//--------------------------------------------------------------------------------------
// Cyclic action
	IF (me.StateMachine.intState=me.StateMachine.intStateLastCycle) THEN
		
		//----------------------------------------------------------------------
		// Substates to let pass hanger(S) from zone 1
		// Triggered by command "Release" (common job interface)
		//----------------------------------------------------------------------		
		CASE me.SubStateMachine.intState OF	
			cSTA_SUB_WAIT_FOR_CMD:
				// Wait for command release
				IF (me.intCmd=STB_CmdState.cCMD_RELEASE) THEN
					CIf.Job.intACmd:=cSTA_DONE;
					me.SubStateMachine.intStateNext := cSTA_SUB_SEND_RELEASE;		
				END_IF
					
			cSTA_SUB_SEND_RELEASE:				
				// Send release command to buffer zone 1
				a_pBufferZoneChildCIF[0]^.Job.intACmd:= STB_CmdState.cCMD_RELEASE;
							
				// State Change Condition
				IF(a_pBufferZoneChildCIF[0]^.Job.intState = STB_CmdState.cSTA_RELEASE)THEN
					me.SubStateMachine.intStateNext := cSTA_SUB_SEND_STOP;					
				END_IF		

			cSTA_SUB_SEND_STOP:
				// Send stop command to buffer zone 1
				a_pBufferZoneChildCIF[0]^.Job.intACmd:= cCMD_STOP;	
				
				// State Change Condition
				IF(a_pBufferZoneChildCIF[0]^.Job.intState = cSTA_STOP)THEN
					me.SubStateMachine.intStateNext := cSTA_SUB_WAIT_FOR_CMD;																
				END_IF	
		
			cSTA_SUB_BREAK:
				//..not used	
		
		END_CASE
				
		
		//----------------------------------------------------------------------
		// Continuous refill of all zones
		//----------------------------------------------------------------------
		
		// Only execute method if more than one buffer zones exist!
		// Note: Slide buffer controller can also used with only one buffer.
		IF (usiNumOfBufferZones>1) THEN				
			THIS^.RefillZones();
		END_IF
			
			
		// Sub state machine general handling
		me.SubStateMachine.intStateLastCycle := me.SubStateMachine.intState;
		CIf.Job.strSubState := THIS^.getCmdState(intCmdState:=me.SubStateMachine.intState,bolState:=TRUE);
		IF (me.SubStateMachine.intState<>me.SubStateMachine.intStateNext) THEN
			me.SubStateMachine.intState := me.SubStateMachine.intStateNext;  // set next state for next cycle
			me.SubStateMachine.udiTimeInState_ms := 0; // reset timer
			// log state change -> open point
		ELSE
			// increment time in state	
			me.SubStateMachine.udiTimeInState_ms := me.SubStateMachine.udiTimeInState_ms + me.FUBInfo.udiSample_ms;
		END_IF
	
		
		// State Change Condition
		IF ((me.intCmd=cCMD_STOP) AND (me.SubStateMachine.intState=cSTA_SUB_WAIT_FOR_CMD))THEN
			me.StateMachine.intStateNext := cSTA_STOPBusy;
		ELSIF ((me.intCmd=STB_CmdState.cCMD_RELEASE_ALL) AND (me.SubStateMachine.intState=cSTA_SUB_WAIT_FOR_CMD))THEN
			me.StateMachine.intStateNext := STB_CmdState.cSTA_RELEASE_ALLBusy;
		END_IF
	END_IF

//--------------------------------------------------------------------------------------
// Exit action
	IF (me.StateMachine.intState<>me.StateMachine.intStateNext) THEN
		;
	END_IF
END_METHOD

METHOD PROTECTED sta_RUNBusy : BOOL
// state implemetation
//--------------------------------------------------------------------------------------
// Entry action
	IF (me.StateMachine.intState<>me.StateMachine.intStateLastCycle) THEN
		me.StateMachine.intStateLastCycle := me.StateMachine.intState;
		
		// Init for refill sequence
		intIndexRefill:= 0;
		SubStateMachineRefill:=0;
	
		// Initialize sub state machine
		me.SubStateMachine.intState:= cSTA_SUB_WAIT_FOR_CMD; 
		me.SubStateMachine.intStateNext := cSTA_SUB_WAIT_FOR_CMD;
	END_IF

	
//--------------------------------------------------------------------------------------
// Cyclic action
	IF (me.StateMachine.intState=me.StateMachine.intStateLastCycle) THEN
			
	
		// State Change Condition	
		IF (TRUE) THEN
			me.StateMachine.intStateNext := cSTA_RUN;		
		END_IF

	END_IF

//--------------------------------------------------------------------------------------
// Exit action
	IF (me.StateMachine.intState<>me.StateMachine.intStateNext) THEN
		;
	END_IF
END_METHOD

METHOD PROTECTED sta_STOP : BOOL
// state implemetation
//--------------------------------------------------------------------------------------
// Entry action
	IF (me.StateMachine.intState<>me.StateMachine.intStateLastCycle) THEN
		me.StateMachine.intStateLastCycle := me.StateMachine.intState;
		;
	END_IF

//--------------------------------------------------------------------------------------
// Cyclic action
	IF (me.StateMachine.intState=me.StateMachine.intStateLastCycle) THEN

	
		// State Change Condition	
		IF (me.intCmd = cCMD_RUN) THEN 
			me.StateMachine.intStateNext := cSTA_RUNBusy;
		ELSIF(me.intCmd = SLB_CmdState.cCMD_RELEASE_ALL) THEN
			me.StateMachine.intStateNext := SLB_CmdState.cSTA_RELEASE_ALLBusy;
		END_IF
	END_IF

//-------------------------------------------------------------------------------------
// Exit action
	IF (me.StateMachine.intState<>me.StateMachine.intStateNext) THEN
		;
	END_IF
END_METHOD

METHOD PROTECTED sta_STOPBusy : BOOL
// state implemetation
//--------------------------------------------------------------------------------------
// Entry action
	IF (me.StateMachine.intState<>me.StateMachine.intStateLastCycle) THEN
		me.StateMachine.intStateLastCycle := me.StateMachine.intState;
		
		// send command STOP to all existing buffer zone child controller.
		THIS^.CmdToAllZones(cCMD_STOP);

	END_IF

//--------------------------------------------------------------------------------------
// Cyclic action
	IF (me.StateMachine.intState=me.StateMachine.intStateLastCycle) THEN
			
				
		// State Change Condition
		// Check if all STOPPED
		IF (THIS^.checkStateAllZones(cSTA_STOP)) THEN
			me.StateMachine.intStateNext := cSTA_STOP;
		END_IF
	END_IF

//--------------------------------------------------------------------------------------
// Exit action
	IF (me.StateMachine.intState<>me.StateMachine.intStateNext) THEN
		;
	END_IF
END_METHOD

METHOD PROTECTED StateMachine : BOOL
SUPER^.StateMachine();

// main statemachine of base controller
CASE me.StateMachine.intState OF
    cSTA_STOPBusy: 
        THIS^.sta_STOPBusy();
    cSTA_STOP: 
        THIS^.sta_STOP();
	cSTA_RUNBusy: 
        THIS^.sta_RUNBusy();
    cSTA_RUN: 
        THIS^.sta_RUN();				
    SLB_CmdState.cSTA_RELEASE_ALLBusy: 
        THIS^.sta_RELEASE_ALLBusy();
    SLB_CmdState.cSTA_RELEASE_ALL: 
        THIS^.sta_RELEASE_ALL();
END_CASE;
END_METHOD

END_FUNCTION_BLOCK

// POUs/Controller/Lvl2/COS (Control Station)/FB_COS
FUNCTION_BLOCK FB_COS EXTENDS FB_CtrlBase
VAR_INPUT
	/// push button next shirt
	In_bolNextShirt: BOOL;
	/// pointer to function block Slide Buffer
	p_fbSLB: POINTER TO FB_SLB;
	/// pointer to function block RFID
	p_fbRFW: POINTER TO FB_RFW;
	/// pointer to function block Single Stopper Buffer
	p_fbSSB: POINTER TO FB_STB;
	/// pointer to function block Drive
	p_fbTLS: POINTER TO FB_DRV;
END_VAR
VAR
	/// Specific interface struct for public access
	SIf: T_Ctrl_SIf_COS;
	/// Interface to Childs
	pSLB_CIF: POINTER TO T_Ctrl_CIf;
	pRFW_CIF: POINTER TO T_Ctrl_CIf;
	pSSB_CIF: POINTER TO T_Ctrl_CIf;
	pTLS_CIF: POINTER TO T_Ctrl_CIf;
	pSLB_SIF: POINTER TO T_Ctrl_SIf_SLB;
	pSSB_SIF: POINTER TO T_Ctrl_SIf_STB;
	/// Function specific variables
	/// edge detection push button
	usi_fpNextShirt: USINT;
END_VAR
VAR CONSTANT
	///sub States for RELEASE Function
	cSTA_SUB_WAIT_FOR_CMD: INT := 500;
	cSTA_SUB_SEND_RELEASE: INT := 501;
	cSTA_SUB_SEND_STOP: INT := 502;
END_VAR

(*__________________________________________________________________________________________________
¦	
¦	Vistaprint Schweiz GmbH
¦	CH - 8401 Winterthur
¦
¦	www.vistaprint.ch - info@vistaprint.ch
¦___________________________________________________________________________________________________

Function desription:
This module manages the flow of the shirts for checking the quality by the operator. 
As soon as the operator presses the button new shirt, the shirt at the operator stopper is released. 
After that the next shirt is released from the slide buffer to the operator stopper. 
The RFID readers communicate all the time the actual controlled shirt to the line controller. 
The ascending conveyor is running the whole time.

History:
Version		Date			Author		Comment
---------------------------------------------------------------------------------------------------
0.00.1		11.09.2013		AVM/KVO		Start history
0.00.2		04.12.2013		AVM/DSC		Input In_bolCounterIn, In_bolCounterOut and In_bolEmergencyOffOk deleted. 
										Handled in parent controller.
0.00.3		10.12.2013		AVM/DSC		Delete condition "me.Alarm.eActivAlmClass=E_AlmClass.STOP" in always method. 
										Don't change to state OFF_busy in case if active alm class is STOP.
0.00.4		16.12.2013		AVM/MRU		Overrule error always from base -> no EOFF State!! in EOFF go to OFF
						
___________________________________________________________________________________________________*)


IF ((me.bolActivate) AND (p_fbSLB<>0) AND (p_fbRFW<>0) AND (p_fbSSB<>0) AND (p_fbTLS<>0)) THEN // cyclic call enabled
	IF (CIf.Info.bolInitDone=FALSE) THEN // first cycle -> init
		CtrlInit();
		CIf.Info.bolInitDone := TRUE;
	ELSE
		CycleStartDuty();
	
		Always();
		
		StateMachine();
		
		CycleEndDuty();
	END_IF
END_IF;

METHOD PROTECTED Always : BOOL
IF (me.bolChangeBackToAUTO=TRUE) THEN // switch mode to automatic switch off controller
	//me.StateMachine.intStateNext := cSTA_OFFBusy;
	//me.bolChangeBackToAUTO := FALSE; // for cylinder no change to off when switch to automatic!!
END_IF

SUPER^.Always();

// ----------------------------------------------------------------------------------
// cyclic actions outside of statemachine
IF (me.StateMachine.intState<>cSTA_SINGLE_ANSWER) THEN
	;
END_IF


// ----------------------------------------------------------------------------------
// Always change actions in Base Library
// ----------------------------------------------------------------------------------
// overrule error always from base -> no EOFF State!! in EOFF go to OFF
IF (me.StateMachine.intStateNext = cSTA_EOFFBusy) THEN
	IF (me.StateMachine.intState=cSTA_OFF) THEN
		me.StateMachine.intStateNext := cSTA_OFF;
	ELSE // stay in OFF
		me.StateMachine.intStateNext := cSTA_OFFBusy;
	END_IF
END_IF

// Conditions Always
IF (((me.Alarm.eActivAlmClass=E_AlmClass.EOFF) OR (me.Alarm.eActivAlmClass=E_AlmClass.OFF) OR (me.intCmd=cCMD_OFF))
		 AND (me.StateMachine.intState<>cSTA_ERROR) AND (me.StateMachine.intState<>cSTA_ERRORQuit) AND
		(me.StateMachine.intState<>cSTA_OFF) AND (me.StateMachine.intState<>cSTA_OFFBusy)) THEN
	// alarm evt EOFF, OFF or cmd off
	me.StateMachine.intStateNext := cSTA_OFFBusy;
END_IF
END_METHOD

METHOD checkChildAlmClass : BOOL
//------------------------------------------------------------------------------------------------------
// check child alarm classes
IF (THIS^.CheckAllChildAlmClass(E_AlmClass.EOFF)) THEN
	CIf.Job.eMe_ActivAlmClass := E_AlmClass.EOFF;
	me.Alarm.bolfp := TRUE;
ELSIF (THIS^.CheckAllChildAlmClass(E_AlmClass.OFF)) THEN
	CIf.Job.eMe_ActivAlmClass := E_AlmClass.OFF;
	me.Alarm.bolfp := TRUE;
ELSIF (THIS^.CheckAllChildAlmClass(E_AlmClass.STOP)) THEN
	CIf.Job.eMe_ActivAlmClass := E_AlmClass.STOP;
	me.Alarm.bolfp := TRUE;
ELSE
	IF (me.Alarm.bolfp) THEN
		CIf.Job.eMe_ActivAlmClass := E_AlmClass.NONE; // no reset necessary
		me.Alarm.bolfp := FALSE;
	END_IF
END_IF

//------------------------------------------------------------------------------------------------------
// set alarm class parent of childs in the case of a parent EOFF or me=OFF or EOFF
IF (CIf.Job.eParent_ActivAlmClass=E_AlmClass.EOFF) THEN
	SetAllChildAlmClass(CIf.Job.eParent_ActivAlmClass);
ELSIF(CIf.Job.eMe_ActivAlmClass=E_AlmClass.EOFF) OR (CIf.Job.eMe_ActivAlmClass=E_AlmClass.OFF) THEN
	SetAllChildAlmClass(CIf.Job.eMe_ActivAlmClass);
ELSE
	// no important alarm for child active
	SetAllChildAlmClass(E_AlmClass.NONE);
END_IF
END_METHOD

METHOD PROTECTED CtrlInit : BOOL
VAR
	ii: INT;
	usiChildIndex: USINT;
END_VAR
SUPER^.CtrlInit();

pSLB_CIF := THIS^.AddChild(p_fbSLB^);
pRFW_CIF := THIS^.AddChild(p_fbRFW^);
pSSB_CIF := THIS^.AddChild(p_fbSSB^);
pTLS_CIF := THIS^.AddChild(p_fbTLS^);

// get specific interface for additional parmaeters or cur
pSLB_SIf := p_fbSLB^.getCtrlSIf();
pSSB_SIf := p_fbSSB^.getCtrlSIf();
//*******************************************************************************
// initial values childes
//*******************************************************************************
END_METHOD

METHOD FB_init : BOOL
VAR_INPUT
	///if TRUE, the retain variables are initialized (warm start / cold start)
	bInitRetains: BOOL;
	///if TRUE, the instance afterwards gets moved into the copy code (online change)
	bInCopyCode: BOOL;
END_VAR
VAR
	udiTaskCnt: UDINT;
	ii: UINT;
END_VAR
//------------------------------------------------------------------------------------------------------------------------
// to manually change in new FUB implementation!!!
// define valid commands for this controller
FOR ii:= 0 TO (SIZEOF(CIf.Job.aCmdList)/SIZEOF(CIf.Job.aCmdList[0])-1) BY 1 DO
	IF (CIf.Job.aCmdList[ii].intCmd=cCMD_INITIALIZED) THEN
		// found first empty array element
		EXIT;
	END_IF
END_FOR
CIf.Job.aCmdList[ii].intCmd := cCMD_RUN;
CIf.Job.aCmdList[ii].strName := 'Run'; 
CIf.Job.aCmdList[ii].bolAvailable := TRUE;
ii := ii +1;
CIf.Job.aCmdList[ii].intCmd := cCMD_STOP;
CIf.Job.aCmdList[ii].strName := 'Stop'; 
CIf.Job.aCmdList[ii].bolAvailable := TRUE;
ii := ii +1;

// set name of class/typ
CIf.Info.strType := 'FB_COS'; 

// set alarm class

//*******************************************************************************
// initial values
//*******************************************************************************

// software configuration
CIf.SwCfg.bolExist := TRUE;
CIf.SwCfg.bolSimulation := FALSE;

// Configuration

// parmeter
END_METHOD

METHOD PROTECTED getCmdState : STRING
VAR_INPUT
	intCmdState: INT;
	bolState: BOOL;
END_VAR
getCmdState := SUPER^.getCmdState(intCmdState:=intCmdState,bolState:=bolState); // get global/base defined cmds/states
IF (getCmdState='') THEN // global not defined get local
	// get string cmd/state string information in runtime
	IF (bolState=FALSE) THEN
		// cmd's
		CASE intCmdState OF
			COS_CmdState.cCMD_RELEASE:
				getCmdState := 'cCMD_RELEASE';
		END_CASE;
	ELSE
	
	// cmd's
		CASE intCmdState OF
			COS_CmdState.cSTA_RELEASEBusy:
				getCmdState := 'cSTA_RELEASEBusy';
			COS_CmdState.cSTA_RELEASE:
				getCmdState := 'cSTA_RELEASE';
				
			// SUB States
			cSTA_SUB_WAIT_FOR_CMD:
				getCmdState := 'cSTA_SUB_WAIT_FOR_CMD';
			cSTA_SUB_SEND_RELEASE:
				getCmdState := 'cSTA_SUB_SEND_RELEASE';
			cSTA_SUB_SEND_STOP:
				getCmdState := 'cSTA_SUB_SEND_STOP';
		END_CASE;
	END_IF
END_IF
END_METHOD

METHOD getCtrlSIf : POINTER TO T_Ctrl_SIf_COS
getCtrlSIf := ADR(SIf);
END_METHOD

METHOD PROTECTED IoInBridge : BOOL
// digitale and analoge inputs read from hardware or forcing
SIf.In.bolNextShirt.map := THIS^.In_bolNextShirt;

IF (CIf.SwCfg.bolSimulation = FALSE) THEN
	getInBol(CIf.Job.bolIoForce,ADR(SIf.In.bolNextShirt));
ELSE
	//simulation of global IO
END_IF
END_METHOD

METHOD PROTECTED sta_OFF : BOOL
// state implemetation
//--------------------------------------------------------------------------------------
// Entry action
	IF (me.StateMachine.intState<>me.StateMachine.intStateLastCycle) THEN
		me.StateMachine.intStateLastCycle := me.StateMachine.intState;

	END_IF


//--------------------------------------------------------------------------------------
// Cyclic action
	IF (me.StateMachine.intState=me.StateMachine.intStateLastCycle) THEN

		// Simulation
		IF (CIf.SwCfg.bolSimulation) THEN
			;
		END_IF
		
		// State Change Condition
		IF ((me.Alarm.eActivAlmClass<>E_AlmClass.EOFF) AND (me.Alarm.eActivAlmClass<>E_AlmClass.OFF)) THEN
			// enable start - no important error active
			IF(me.intCmd=cCMD_RUN) THEN
				me.StateMachine.intStateNext := cSTA_RUNBusy;
			END_IF
		END_IF
	END_IF




//--------------------------------------------------------------------------------------
// Exit action
	IF (me.StateMachine.intState<>me.StateMachine.intStateNext) THEN
		;
	END_IF
END_METHOD

METHOD PROTECTED sta_RUN : BOOL
// state implemetation
//--------------------------------------------------------------------------------------
// Entry action
	IF (me.StateMachine.intState<>me.StateMachine.intStateLastCycle) THEN
		me.StateMachine.intStateLastCycle := me.StateMachine.intState;
		
		me.SubStateMachine.intState := cSTA_SUB_WAIT_FOR_CMD; // init sub state machine
		me.SubStateMachine.intStateNext := cSTA_SUB_WAIT_FOR_CMD; // init sub state machine

	END_IF


//--------------------------------------------------------------------------------------
// Cyclic action
	IF (me.StateMachine.intState=me.StateMachine.intStateLastCycle) THEN

		// Simulation
		IF (CIf.SwCfg.bolSimulation) THEN
			;
		END_IF

		// positive edge detect -> release next shirt
		IF (SIf.In.bolNextShirt.intern=1) THEN
			IF (usi_fpNextShirt=0) THEN 
				usi_fpNextShirt := 1;
			END_IF
		ELSE
			usi_fpNextShirt := 0;
		END_IF
		
		CASE me.SubStateMachine.intState OF	
		// Start Cycle with substates	
		//--------------------------------------------------------------------------------------
		// sub state machine for sequence
		cSTA_SUB_WAIT_FOR_CMD:
		
			// Wait for command next shirt
			IF (usi_fpNextShirt=1) THEN
				usi_fpNextShirt := 2;
				me.SubStateMachine.intStateNext := cSTA_SUB_SEND_RELEASE;		
			ELSIF (me.intCmd=STB_CmdState.cCMD_RELEASE) THEN
				CIf.Job.intACmd:=cSTA_DONE;
				me.SubStateMachine.intStateNext := cSTA_SUB_SEND_RELEASE;		
			END_IF	
			
		cSTA_SUB_SEND_RELEASE:				
			// Send release command to single stopper
			pSSB_CIF^.Job.intACmd:= STB_CmdState.cCMD_RELEASE;

			// State Change Condition
			IF(pSSB_CIF^.Job.intState = STB_CmdState.cSTA_RELEASE)THEN
				me.SubStateMachine.intStateNext := cSTA_SUB_SEND_STOP;	
				pSLB_CIF^.Job.intACmd:= SLB_CmdState.cCMD_RELEASE;				
			END_IF		

		cSTA_SUB_SEND_STOP:
			// Send stop command to single stopper
			pSSB_CIF^.Job.intACmd:= cCMD_STOP;	
			
			// State Change Condition
			IF (pSSB_CIF^.Job.intState = cSTA_STOP) AND (CIf.Job.intACmd = cSTA_DONE)THEN
				me.SubStateMachine.intStateNext := cSTA_SUB_WAIT_FOR_CMD;																
			END_IF

		END_CASE
		
		me.SubStateMachine.intStateLastCycle := me.SubStateMachine.intState;
		CIf.Job.strSubState := THIS^.getCmdState(intCmdState:=me.SubStateMachine.intState,bolState:=TRUE);
		IF (me.SubStateMachine.intState<>me.SubStateMachine.intStateNext) THEN
			me.SubStateMachine.intState := me.SubStateMachine.intStateNext;  // set next state for next cycle
			me.SubStateMachine.udiTimeInState_ms := 0; // reset timer
			// log state change -> open point
		ELSE
			// increment time in state	
			me.SubStateMachine.udiTimeInState_ms := me.SubStateMachine.udiTimeInState_ms + me.FUBInfo.udiSample_ms;
		END_IF
				
		// State Change Condition	
		IF (me.intCmd=cCMD_STOP) THEN
			me.StateMachine.intStateNext :=  cSTA_STOPBusy;	
		END_IF
	END_IF

//--------------------------------------------------------------------------------------
// Exit action
	IF (me.StateMachine.intState<>me.StateMachine.intStateNext) THEN
		;
	END_IF
END_METHOD

METHOD PROTECTED sta_RUNBusy : BOOL
// state implemetation
//--------------------------------------------------------------------------------------
// Entry action
	IF (me.StateMachine.intState<>me.StateMachine.intStateLastCycle) THEN
		me.StateMachine.intStateLastCycle := me.StateMachine.intState;
		
	END_IF


//--------------------------------------------------------------------------------------
// Cyclic action
	IF (me.StateMachine.intState=me.StateMachine.intStateLastCycle) THEN

		// Simulation
		
		// Cyclic action
		pSLB_CIF^.Job.intACmd := cCMD_RUN;
		pRFW_CIF^.Job.intACmd := cCMD_RUN;
		
		IF ( (pSLB_CIF^.Job.intState = cSTA_RUN) AND (pRFW_CIF^.Job.intState = cSTA_RUN))  THEN
			pTLS_CIF^.Job.intACmd := cCMD_RUN;
			pSSB_CIF^.Job.intACmd := cCMD_STOP;
		END_IF;

		// State Change Condition
		IF ( (pSLB_CIF^.Job.intState = cSTA_RUN) AND (pRFW_CIF^.Job.intState = cSTA_RUN) AND
			(pSSB_CIF^.Job.intState = cSTA_STOP) AND (pTLS_CIF^.Job.intState = cSTA_RUN))  THEN
			me.StateMachine.intStateNext := cSTA_RUN;
		ELSIF (me.intCmd=cCMD_STOP) THEN
			me.StateMachine.intStateNext :=  cSTA_STOPBusy;	
		END_IF
	END_IF




//--------------------------------------------------------------------------------------
// Exit action
	IF (me.StateMachine.intState<>me.StateMachine.intStateNext) THEN
		;
	END_IF
END_METHOD

METHOD PROTECTED sta_STOP : BOOL
// state implemetation
//--------------------------------------------------------------------------------------
// Entry action
	IF (me.StateMachine.intState<>me.StateMachine.intStateLastCycle) THEN
		me.StateMachine.intStateLastCycle := me.StateMachine.intState;
		
	END_IF


//--------------------------------------------------------------------------------------
// Cyclic action
	IF (me.StateMachine.intState=me.StateMachine.intStateLastCycle) THEN
		
		;
		
		
		// State Change Condition
		IF (me.intCmd=cCMD_RUN) THEN
			me.StateMachine.intStateNext :=  cSTA_RUNBusy;
		END_IF
	END_IF




//--------------------------------------------------------------------------------------
// Exit action
	IF (me.StateMachine.intState<>me.StateMachine.intStateNext) THEN
		;
	END_IF
END_METHOD

METHOD PROTECTED sta_STOPBusy : BOOL
// state implemetation
//--------------------------------------------------------------------------------------
// Entry action
	IF (me.StateMachine.intState<>me.StateMachine.intStateLastCycle) THEN
		me.StateMachine.intStateLastCycle := me.StateMachine.intState;
		

	END_IF


//--------------------------------------------------------------------------------------
// Cyclic action
	IF (me.StateMachine.intState=me.StateMachine.intStateLastCycle) THEN

		// Simulation
		IF (CIf.SwCfg.bolSimulation) THEN
			;
		END_IF
		
		// Cyclicle action
		pSLB_CIF^.Job.intACmd := cCMD_STOP;

		IF (pSLB_CIF^.Job.intState = cCMD_STOP)  THEN
			pTLS_CIF^.Job.intACmd := cCMD_OFF;
			pSSB_CIF^.Job.intACmd := cCMD_STOP;
		END_IF;

		// State Change Condition
		IF ( (pSLB_CIF^.Job.intState = cSTA_STOP) AND (pSSB_CIF^.Job.intState = cSTA_STOP) AND (pTLS_CIF^.Job.intState = cSTA_OFF))  THEN
			me.StateMachine.intStateNext := cSTA_STOP;
		ELSIF (me.intCmd=cCMD_RUN) THEN
			me.StateMachine.intStateNext :=  cSTA_RUNBusy;	
		END_IF
	END_IF




//--------------------------------------------------------------------------------------
// Exit action
	IF (me.StateMachine.intState<>me.StateMachine.intStateNext) THEN
		;
	END_IF
END_METHOD

METHOD PROTECTED StateMachine : BOOL
SUPER^.StateMachine();

// main statemachine of base controller
CASE me.StateMachine.intState OF
    cSTA_RUNBusy: 
        THIS^.sta_RUNBusy();
    cSTA_RUN: 
        THIS^.sta_RUN();
    cSTA_STOPBusy: 
        THIS^.sta_STOPBusy();
    cSTA_STOP: 
        THIS^.sta_STOP();		
END_CASE;
END_METHOD

END_FUNCTION_BLOCK

// POUs/Controller/Lvl2/FOL (Folder)/FB_FOL
FUNCTION_BLOCK FB_FOL EXTENDS FB_CtrlBase
VAR_INPUT
	p_fbSLB: POINTER TO FB_SLB;
	/// CAN communication to folder
	p_fbFOC: POINTER TO FB_FOC;
	p_fbRFW: POINTER TO FB_RFW;
	p_fbTLS: POINTER TO FB_DRV;
END_VAR
VAR
	/// Specific interface struct for public access
	SIf: T_Ctrl_SIf_FOL;
	/// Child controller
	pSLB_CIf: POINTER TO T_Ctrl_CIf;
	/// CAN communication to folder
	pFOC_CIf: POINTER TO T_Ctrl_CIf;
	pRFW_CIf: POINTER TO T_Ctrl_CIf;
	pTLS_CIf: POINTER TO T_Ctrl_CIf;
	pSLB_SIF: POINTER TO T_Ctrl_SIf_SLB;
END_VAR
VAR CONSTANT
	cSTA_SUB_INITIALIZED: INT := 500;
	cSTA_SUB_START_ELEMENTS: INT := 502;
	cSTA_SUB_START_CYCLE: INT := 504;
	cSTA_SUB_START_WAIT_CYCLE: INT := 506;
	cSTA_SUB_START_FINAL: INT := 511;
	cSTA_SUB_FINISHED: INT := 600;
END_VAR

(*__________________________________________________________________________________________________
¦	
¦	Vistaprint Schweiz GmbH
¦	CH - 8401 Winterthur
¦
¦	www.vistaprint.ch - info@vistaprint.ch
¦___________________________________________________________________________________________________

Function desription:
Folder module instance controls Folder robot, slide buffer before folder, TLS conveyor for empty hangers and RFID reader in Folder.


History:
Version		Date			Author		Comment
---------------------------------------------------------------------------------------------------
0.00.1		01.10.2013		VP/RE		Start history
0.00.2		11.12.2013		AVME/MRU	Add Methode checkChildAlmClass for Error Stop of childs

___________________________________________________________________________________________________*)


// check if child pointer valid
IF ((me.bolActivate) AND (p_fbSLB<>0) AND (p_fbRFW<>0) AND (p_fbTLS<>0)) THEN // cyclic call enabled
	
	IF (CIf.Info.bolInitDone=FALSE) THEN // first cycle -> init
		CtrlInit();
		CIf.Info.bolInitDone := TRUE;
	ELSE
		CycleStartDuty();
	
		Always();
		
		StateMachine();
		
		CycleEndDuty();
	END_IF
	
END_IF;

METHOD PROTECTED Always : BOOL
IF (me.bolChangeBackToAUTO=TRUE) THEN // switch mode to automatic switch off controller
	//me.StateMachine.intStateNext := cSTA_OFFBusy;
	//me.bolChangeBackToAUTO := FALSE; // for cylinder no change to off when switch to automatic!!
END_IF

SUPER^.Always();

// ----------------------------------------------------------------------------------
// cyclic actions outside of statemachine
IF (me.StateMachine.intState<>cSTA_SINGLE_ANSWER) THEN
	;
END_IF

SIf.Cur.dinMaxCapacity := p_fbSLB^.getCtrlSIf()^.Cur.dinMaxCapacity;
SIf.Cur.bolIsFull := p_fbSLB^.getCtrlSIf()^.Cur.bolInputBufferFull;

// ----------------------------------------------------------------------------------
// Conditions Always
// overrule error always from base -> no EOFF State!! in EOFF go to OFF
IF (me.StateMachine.intStateNext = cSTA_EOFFBusy) THEN
	IF (me.StateMachine.intState=cSTA_OFF) THEN
		me.StateMachine.intStateNext := cSTA_OFF;
	ELSE // stay in OFF
		me.StateMachine.intStateNext := cSTA_OFFBusy;
	END_IF
END_IF
END_METHOD

METHOD checkChildAlmClass : BOOL
//------------------------------------------------------------------------------------------------------
// check child alarm classes
// set me alarm class active if at least one child has an EOFF
IF CheckAllChildAlmClass(E_AlmClass.EOFF) THEN
	CIf.Job.eMe_ActivAlmClass := E_AlmClass.EOFF;
	me.Alarm.bolfp := TRUE;
ELSIF CheckAllChildAlmClass(E_AlmClass.OFF) THEN
	CIf.Job.eMe_ActivAlmClass := E_AlmClass.OFF;
	me.Alarm.bolfp := TRUE;
ELSIF CheckAllChildAlmClass(E_AlmClass.STOP) THEN  // FB_MER needs alarm class STOP
	CIf.Job.eMe_ActivAlmClass := E_AlmClass.STOP;
	me.Alarm.bolfp := TRUE;
ELSE
	IF (me.Alarm.bolfp) THEN
		CIf.Job.eMe_ActivAlmClass := E_AlmClass.NONE; // no reset necessary
		me.Alarm.bolfp := FALSE;
	END_IF
END_IF

//------------------------------------------------------------------------------------------------------
// set alarm class parent of childs
//------------------------------------------------------------------------------------------------------
// set alarm class parent of childs in the case of a parent EOFF or me=OFF or EOFF
IF (CIf.Job.eParent_ActivAlmClass=E_AlmClass.EOFF) THEN
	SetAllChildAlmClass(CIf.Job.eParent_ActivAlmClass);
ELSIF(CIf.Job.eMe_ActivAlmClass=E_AlmClass.EOFF) OR (CIf.Job.eMe_ActivAlmClass=E_AlmClass.OFF) THEN
	SetAllChildAlmClass(CIf.Job.eMe_ActivAlmClass);
ELSE
	// no important alarm for child active
	SetAllChildAlmClass(E_AlmClass.NONE);
END_IF
END_METHOD

METHOD PROTECTED CtrlInit : BOOL
SUPER^.CtrlInit();

// get child CIf
pSLB_CIf := THIS^.AddChild(p_fbSLB^);
pFOC_CIf := THIS^.AddChild(p_fbFOC^);
pRFW_CIf := THIS^.AddChild(p_fbRFW^);
pTLS_CIf := THIS^.AddChild(p_fbTLS^);

pSLB_SIF := p_fbSLB^.getCtrlSIf();
END_METHOD

METHOD FB_init : BOOL
VAR_INPUT
	///if TRUE, the retain variables are initialized (warm start / cold start)
	bInitRetains: BOOL;
	///if TRUE, the instance afterwards gets moved into the copy code (online change)
	bInCopyCode: BOOL;
END_VAR
VAR
	ii: UINT;
END_VAR
//------------------------------------------------------------------------------------------------------------------------
// to manually change in new FUB implementation!!!
// define valid commands for this controller
FOR ii:= 0 TO (SIZEOF(CIf.Job.aCmdList)/SIZEOF(CIf.Job.aCmdList[0])-1) BY 1 DO
	IF (CIf.Job.aCmdList[ii].intCmd=cCMD_INITIALIZED) THEN
		// found first empty array element
		EXIT;
	END_IF
END_FOR
CIf.Job.aCmdList[ii].intCmd := cCMD_RUN;
CIf.Job.aCmdList[ii].strName := 'Run'; 
CIf.Job.aCmdList[ii].bolAvailable := TRUE;
//ii := ii +1;
//CIf.Job.aCmdList[ii].intCmd := cCMD_RETRACT;
//CIf.Job.aCmdList[ii].strName := 'Retract';
//CIf.Job.aCmdList[ii].bolAvailable := TRUE;

// set name of class/typ
CIf.Info.strType := 'FB_FOL'; 

// set alarm class
SIf.Alm[1].eAlmClass := E_AlmClass.INFO;
SIf.Alm[1].strText := 'Reserve'; 

//*******************************************************************************
// initial values
//*******************************************************************************

// software configuration
CIf.SwCfg.bolExist := TRUE;
CIf.SwCfg.bolSimulation := FALSE;

// parmeter
//SIf.Par.udiDelayFirstClamp_ms := 750;

// actual values
//SIf.Cur.dinCounter := 0;
END_METHOD

METHOD PROTECTED getCmdState : STRING
VAR_INPUT
	intCmdState: INT;
	bolState: BOOL;
END_VAR
getCmdState := SUPER^.getCmdState(intCmdState:=intCmdState,bolState:=bolState); // get global/base defined cmds/states

IF (getCmdState='') THEN // global not defined get local
	// get string cmd/state string information in runtime
	IF (bolState=FALSE) THEN
		// cmd's
	ELSE
	
	// cmd's
		CASE intCmdState OF
				
			// SUB States
			cSTA_SUB_INITIALIZED:
				getCmdState := 'cSTA_SUB_INITIALIZED';
			cSTA_SUB_START_CYCLE:
				getCmdState := 'cSTA_SUB_START_CYCLE';
			cSTA_SUB_START_Wait_CYCLE:
				getCmdState := 'cSTA_SUB_START_Wait_CYCLE';
			cSTA_SUB_START_ELEMENTS:
				getCmdState := 'cSTA_SUB_START_ELEMENTS';
			cSTA_SUB_START_FINAL:
				getCmdState := 'cSTA_SUB_START_FINAL';
			cSTA_SUB_FINISHED:
				getCmdState := 'cSTA_SUB_FINISHED';
		END_CASE;
	END_IF
END_IF
END_METHOD

METHOD getCtrlSIf : POINTER TO T_Ctrl_SIf_FOL
getCtrlSIf := ADR(SIf);
END_METHOD

METHOD PROTECTED IoInBridge : BOOL
// digitale and analoge inputs read from hardware or forcing
//SIf.In.bolEmergencyStop.map := THIS^.In_EmergencyStop;

IF (CIf.SwCfg.bolSimulation = FALSE) THEN
	//getInBol(CIf.Job.bolIoForce,ADR(SIf.In.bolEmergencyStop));
ELSE
	//simulation of global IO
END_IF
END_METHOD

METHOD PROTECTED IoOutBridge : BOOL
VAR
	bolSwitchValvesOff: BOOL;
END_VAR
// digitale and analoge inputs read from hardware or forcing
IF (CIf.SwCfg.bolSimulation = FALSE) THEN
//	setOutBol(CIf.Job.bolIoForce ,ADR(SIf.Out.bolClamping));

//	THIS^.Out_Clamping := SIf.Out.bolClamping.map;
END_IF
END_METHOD

METHOD PROTECTED sta_OFF : BOOL
// state implemetation
//--------------------------------------------------------------------------------------
// Entry action
	IF (me.StateMachine.intState<>me.StateMachine.intStateLastCycle) THEN
		me.StateMachine.intStateLastCycle := me.StateMachine.intState;
		
	END_IF

//--------------------------------------------------------------------------------------
// Cyclic action
	IF (me.StateMachine.intState=me.StateMachine.intStateLastCycle) THEN
				
		// State Change Condition
		IF ((me.Alarm.eActivAlmClass<>E_AlmClass.EOFF) AND (me.Alarm.eActivAlmClass<>E_AlmClass.OFF)) THEN
			// enable start - no important error active
			IF me.intCmd=cCMD_RUN THEN
				me.StateMachine.intStateNext :=  cSTA_RUNBusy;
			END_IF
		END_IF
	END_IF


//--------------------------------------------------------------------------------------
// Exit action
	IF (me.StateMachine.intState<>me.StateMachine.intStateNext) THEN
		;
	END_IF
END_METHOD

METHOD PROTECTED sta_RUN : BOOL
// state implemetation
//--------------------------------------------------------------------------------------
// Entry action
	IF (me.StateMachine.intState<>me.StateMachine.intStateLastCycle) THEN
		me.StateMachine.intStateLastCycle := me.StateMachine.intState;
	
		me.SubStateMachine.intState := cSTA_SUB_START_CYCLE; // init sub state machine
		me.SubStateMachine.intStateNext := cSTA_SUB_START_CYCLE; // init sub state machine		
	END_IF

//--------------------------------------------------------------------------------------
// Cyclic action
	IF (me.StateMachine.intState=me.StateMachine.intStateLastCycle) THEN

		// Simulation
		IF (CIf.SwCfg.bolSimulation) THEN
			;
		END_IF

		// sub state machine for sequence
		CASE me.SubStateMachine.intState OF

			cSTA_SUB_START_CYCLE:	
				IF (pSLB_SIF^.Cur.bolHangerDetected) THEN
					pSLB_CIf^.Job.intACmd := SLB_CmdState.cCMD_RELEASE;
					me.SubStateMachine.intStateNext := cSTA_SUB_FINISHED;
				END_IF
			
			cSTA_SUB_FINISHED:	
				// Wait until job done
				IF(pSLB_CIf^.Job.intACmd = cSTA_DONE)THEN	
					IF (me.SubStateMachine.udiTimeInState_ms >= SIf.Par.udiTimeNextHangers_ms) THEN
						me.SubStateMachine.intStateNext := cSTA_SUB_START_CYCLE;
					END_IF
				END_IF	
		END_CASE

		// State Change Condition	
		IF (me.intCmd=BASE_PLC.cCMD_OFF) THEN
			me.StateMachine.intStateNext :=  cSTA_OFFBusy;	
		END_IF
	END_IF

//--------------------------------------------------------------------------------------
// Exit action
	IF (me.StateMachine.intState<>me.StateMachine.intStateNext) THEN
		;
	END_IF
END_METHOD

METHOD PROTECTED sta_RUNBusy : BOOL
// state implemetation
//--------------------------------------------------------------------------------------
// Entry action
	IF (me.StateMachine.intState<>me.StateMachine.intStateLastCycle) THEN
		me.StateMachine.intStateLastCycle := me.StateMachine.intState;
		
		me.SubStateMachine.intState := cSTA_SUB_INITIALIZED; // init sub state machine
		me.SubStateMachine.intStateNext := cSTA_SUB_INITIALIZED; // init sub state machine
	END_IF

//--------------------------------------------------------------------------------------
// Cyclic action
	IF (me.StateMachine.intState=me.StateMachine.intStateLastCycle) THEN

		// Simulation
		IF (CIf.SwCfg.bolSimulation) THEN
			fbSimulationTimer(); // simulation time
			IF (fbSimulationTimer.Q) THEN
				;
			END_IF
		END_IF
		
		// Cyclicle action
		// Start Cycle with substates	
		//--------------------------------------------------------------------------------------
		// sub state machine for sequence
		CASE me.SubStateMachine.intState OF
			//--------------------------------------------------------------------------------------
			cSTA_SUB_INITIALIZED:
				me.SubStateMachine.intStateNext := cSTA_SUB_START_ELEMENTS;
				
			cSTA_SUB_START_ELEMENTS:
				//start all childs
				pSLB_CIf^.Job.intACmd := cCMD_RUN;
				pFOC_CIf^.Job.intACmd := cCMD_RUN;
				pRFW_CIf^.Job.intACmd := cCMD_RUN;
				pTLS_CIf^.Job.intACmd := cCMD_RUN;
	
				IF ((pSLB_CIf^.Job.intState = cSTA_RUN) AND (pRFW_CIf^.Job.intState = cSTA_RUN) AND (pTLS_CIf^.Job.intState = cSTA_RUN) AND (pFOC_CIf^.Job.intState = cSTA_RUN)) THEN
					me.SubStateMachine.intStateNext := cSTA_SUB_FINISHED;
				END_IF
				
		//--------------------------------------------------------------------------------------
			cSTA_SUB_FINISHED:
					;
					
		END_CASE
			
		// State Change Condition
		IF (me.SubStateMachine.intState = cSTA_SUB_FINISHED) THEN
			me.StateMachine.intStateNext := cSTA_RUN;
		ELSIF (me.intCmd=cCMD_STOP) THEN
			me.StateMachine.intStateNext :=  cSTA_STOPBusy;	
		END_IF
	END_IF

//--------------------------------------------------------------------------------------
// Exit action
	IF (me.StateMachine.intState<>me.StateMachine.intStateNext) THEN
		;
	END_IF
END_METHOD

METHOD PROTECTED StateMachine : BOOL
SUPER^.StateMachine();

// main statemachine of base controller
CASE me.StateMachine.intState OF
    cSTA_RUNBusy: 
        THIS^.sta_RUNBusy();
    cSTA_RUN: 
        THIS^.sta_RUN();
END_CASE;
END_METHOD

END_FUNCTION_BLOCK

// POUs/Controller/Lvl2/MER (Merger)/FB_MER
FUNCTION_BLOCK FB_MER EXTENDS FB_CtrlBase IMPLEMENTS IBuffer
VAR_INPUT
	// Sensor hanger detected
	In_bolHangerDetected: BOOL;
	// Pin of Drive is detected
	In_bolPinDetected: BOOL;
	// Sensors for jam detection
	In_a_bolJamSensor: ARRAY[1..cMAX_JAM_SENSORS] OF BOOL;
END_VAR
VAR
	// Specific interface struct for public access
	SIf: T_Ctrl_SIf_MER;
	// List of pointers to Childs
	a_pLineChildCtrl: ARRAY[0..Base_Const.cMaxNrOfChilds] OF POINTER TO FB_SLB;
	// List of childs common interface
	a_pLineChildCIF: ARRAY[0..Base_Const.cMaxNrOfChilds] OF POINTER TO T_Ctrl_CIf;
	// List of childs specific interface for additional parameters or cur
	a_pLineChildSIF: ARRAY[0..Base_Const.cMaxNrOfChilds] OF POINTER TO T_Ctrl_SIf_SLB;
	// Function specific variables
	usiNumOfLines: USINT;
	usiNumOfValidPointerToLine: USINT;
	bolHangerExist: BOOL;
	bolGoToRun: BOOL;
	dinPassedTotalLineXOld: DINT;
	// Used for counting passed hangers if "E_Typ_MER_MODE.MergeOverSetpoint" is selected.
	dinNumOfPassedHangers: DINT;
	// Used for time measurement if "E_Typ_MER_MODE.MergeOverTime" is selected.
	udiMergingTime: UDINT;
	usiLineNumToReleaseAll: USINT;
	usiIndexToRelease: USINT;
	// Last new position value from parent
	dinTransportPositionOld_um: DINT;
	// Driven Way in the task
	dinDrivenWay_um: DINT;
	// Position correction in faster Task cycletime
	dinPositionCorrection_um: DINT;
	// Position of the section
	dinPositionSection_um: DINT;
	// Section buffer
	a_stSectionBuffer: ARRAY[0..cusiSectionBuffer_SIZE] OF T_MER_Buffer_Sections;
	// Edge detection of the inputs
	bolRE_HangerDetected: BOOL;
	// Pin of Drive is detected
	bolRE_PinDetected: BOOL;
	bolModeMergeIntoTrpUsed: BOOL;
	bolSectionFree: BOOL;
	bolReleaseHanger: BOOL;
	// Used to detect if a section is driven out
	dinPositionOfLastLine_um: DINT;
	// Shadow copy of In_a_bolJamSensor[]
	a_bolJamSensorOnce: ARRAY[1..cMAX_JAM_SENSORS] OF BOOL;
	// Start time of jam sensor is true
	a_udiTimeJamDetection: ARRAY[1..cMAX_JAM_SENSORS] OF UDINT;
	// Jam release delay timer
	udiJamReleaseDelayTime_ms: UDINT;
	// Jam at merger output detected 
	bolJamDetected: BOOL;
	// Loop variable
	intI: INT;
	// Simulated section length
	dinSimSectionLength_um: DINT := 510000;
	// Simulated way to trigger section start/end
	dinSimWayTrigSection_um: DINT;
END_VAR
VAR CONSTANT
	// sub States
	cSTA_SUB_INITIALIZED: INT := 500;
	cSTA_SUB_WAIT_FOR_CMD: INT := 502;
	cSTA_SUB_CHECK_HANGER_EXIST: INT := 504;
	cSTA_SUB_SEND_RELEASE: INT := 506;
	cSTA_SUB_SEND_RELEASE_ALL: INT := 508;
	cSTA_SUB_SEND_STOP: INT := 510;
	cSTA_SUB_WAIT_JOB_DONE: INT := 512;
	cSTA_SUB_CHECK_MERGE_CON: INT := 514;
	cSTA_SUB_WAIT_LINE_FREE: INT := 516;
	cSTA_SUB_END: INT := 518;
END_VAR

(*__________________________________________________________________________________________________
¦	
¦	Vistaprint Schweiz GmbH
¦	CH - 8401 Winterthur
¦
¦	www.vistaprint.ch - info@vistaprint.ch
¦___________________________________________________________________________________________________

Function desription:
The controller automatically merge hangers from different lines dependent time or distribution of the number of hangers.
Lines are always from controller type slide buffer FB_SLB.

History:
Version		Date			Author		Comment
---------------------------------------------------------------------------------------------------
0.00.1		05.09.2013		AVME/DSC	Start history. 
0.00.2		09.09.2013		AVME/DSC 	Integration of all merger basic functionalities. Test on simulator.
										Controller can work in 2 different main modes:
										-> "automatic", controller automatically merge hangers from different lines dependent E_Typ_MER_AUTO_MODE
										-> "on command", in case if merger work as charge controller. Release line X dependent from parent command.
0.00.3		19.09.2013		AVME/PRE	Implement new Base Concept
0.00.4		01.10.2013		AVME/DSC	Sub state machine general handling deleted. Not used anymore. Handled in Base Class.										
0.00.5		03.10.2013		AVME/PRE	Integrate new function insert Belt		
0.00.6		03.10.2013		AVME/PRE	Insert new sub state LOCK_SECTION.	
0.00.7		15.10.2013		AVME/DSC	Complete redesign of the merger "MergeIntoTrp" mode.
0.00.8		30.10.2013		AVME/DSC	Modifications for "MergeIntoTrp" mode during test at the tool. Good merging possible with drive speed = 0. (slow speed)
										Merging with higher speed not possible!				
0.00.9		08.11.2013		AVME/MRU	Stop merger if outfeed sensor detect a jam (Bugzilla Nr. 8)
0.00.10		03.12.2013		AVME/MRU	Add MaxCapacity / NumOfHangers properties
0.00.11		09.12.2013		AVME/DSC	Modification in method "checkStateAllLines".
										Special condition: In case if the child is in state ERROR and STOP is requested. Set child as checked.
										Parent controller need state STOP that automatic stop sequence can work for all other childs.
0.00.12		13.01.2014		AVME/MRU	Bugzilla ID 03: BufferFull for LineControl added
0.00.13		22.01.2014		AVME/MRU	udiJamReleaseDelayTime_ms added; Timing "Check jam detection" reworked

__________________________________________________________________________________________________*)


IF ((me.bolActivate) AND (THIS^.checkChildValid())) THEN // cyclic call enabled
	IF (CIf.Info.bolInitDone=FALSE) THEN // first cycle -> init
		CtrlInit();
		CIf.Info.bolInitDone := TRUE;
	ELSE
		CycleStartDuty();
	
		Always();
		
		StateMachine();
		
		CycleEndDuty();
	END_IF
END_IF;

METHOD AddLine
VAR_INPUT
	p_Line: POINTER TO FB_SLB;
END_VAR

// Method add the pointer address of the line child controller to the array list.
IF (usiNumOfLines <= (Base_Const.cMaxNrOfChilds-1)) THEN
	// Add line child controller to list
	a_pLineChildCtrl[usiNumOfLines] := p_Line;
	// Inc. number of lines
	usiNumOfLines:= usiNumOfLines+1;
	// Check if the pointer is valid
	IF (p_Line<>0) THEN
		usiNumOfValidPointerToLine:= usiNumOfValidPointerToLine+1;
	END_IF
END_IF
END_METHOD

METHOD PROTECTED Always : BOOL
VAR
	/// Looping variable
	intSec: INT;
END_VAR
IF (me.bolChangeBackToAUTO=TRUE) THEN // switch mode to automatic switch off controller
	//me.StateMachine.intStateNext := cSTA_OFFBusy;
	//me.bolChangeBackToAUTO := FALSE; // for cylinder no change to off when switch to automatic!!
END_IF

SUPER^.Always();

// ----------------------------------------------------------------------------------
// cyclic actions outside of statemachine
IF (me.StateMachine.intState<>cSTA_SINGLE_ANSWER) THEN
	
	//-------------------------------------------------
	// Provide current values for the parent
	//-------------------------------------------------	
	
	// Number of lines to merge, depends on how many times the method "AddLine" was called at init
	SIf.Cur.usiNumOfLinesToMerge:= usiNumOfLines;
	// Actual Item Count of this controller -> based on all lines
	SIf.Cur.dinCurrentItemCount:= THIS^.CalcSumOfItems();
	// Max. buffer capacity -> based on all lines
	SIf.Cur.dinMaxCapacity:= THIS^.CalcMaxCapacity();	
	
	
	// Check if mode "MergeIntoTrp" is configured. 
	// If one line is configured with this mode, all other lines will be set to the same mode automatically in CtrlInit. Mixed mode not possible.
	IF ((SIf.Cfg.usiMergeMainMode = E_Typ_MER_MODE.Automatic) AND (SIf.Par.a_LinePar[0].usiMergeMode = E_Typ_MER_AUTO_MODE.MergeIntoTrp)) THEN
	
		//----------------------------------------------------------------------
		// Calculate position for transport 
		//----------------------------------------------------------------------
			
		// If this task is used in a faster cycle as the parent, the driven way will be indirectly calculated (synchronized) over the transport speed.
		// If transport position changed from the parent (new value), synchronize the driven way 
		
		IF (dinTransportPositionOld_um <> SIf.Cur.dinTransportPosition_um) THEN
			dinDrivenWay_um := SIf.Cur.dinTransportPosition_um - SIf.Cur.dinTransportPositionCalc_um;
			SIf.Cur.dinTransportPositionCalc_um := SIf.Cur.dinTransportPosition_um;
			dinTransportPositionOld_um := SIf.Cur.dinTransportPosition_um;
			dinPositionCorrection_um := 0;
		ELSE
			// During the time, if there is no position change from the parent, calculate the driven way dependent the speed of transport.		
			// s = v * t
			dinDrivenWay_um := LREAL_TO_DINT(DINT_TO_LREAL(SIf.Cur.dinTransportspeed_um_s) * UDINT_TO_LREAL(me.FUBInfo.udiSample_ms) / 1000.0 );
			dinPositionCorrection_um := dinPositionCorrection_um + dinDrivenWay_um;
			SIf.Cur.dinTransportPositionCalc_um := dinTransportPositionOld_um + dinPositionCorrection_um;
		END_IF
	
	END_IF
	
END_IF

// ----------------------------------------------------------------------------------
// Always change actions in Base Library
// ----------------------------------------------------------------------------------
// overrule error always from base -> no EOFF State!! in EOFF go to OFF
IF (me.StateMachine.intStateNext = cSTA_EOFFBusy) THEN
	IF (me.StateMachine.intState=cSTA_OFF) THEN
		me.StateMachine.intStateNext := cSTA_OFF;
	ELSE // stay in OFF
		me.StateMachine.intStateNext := cSTA_OFFBusy;
	END_IF
END_IF

// Conditions Always
IF (((me.Alarm.eActivAlmClass=E_AlmClass.EOFF) OR (me.Alarm.eActivAlmClass=E_AlmClass.OFF) OR (me.intCmd=cCMD_OFF))
		 AND (me.StateMachine.intState<>cSTA_ERROR) AND (me.StateMachine.intState<>cSTA_ERRORQuit) AND
		(me.StateMachine.intState<>cSTA_OFF) AND (me.StateMachine.intState<>cSTA_OFFBusy)) THEN
	// alarm evt EOFF, OFF or cmd off
	me.StateMachine.intStateNext := cSTA_OFFBusy;
END_IF
END_METHOD

PROPERTY BufferFull : BOOL
GET
BufferFull:= False;
END_GET
END_PROPERTY

METHOD PROTECTED CalcMaxCapacity : DINT
VAR
	ii: INT;
	dinSumMaxCapacity: DINT;
END_VAR
// Method calculate the sum of max. capacities from all lines and return the result.

//Init
CalcMaxCapacity:= 0;
dinSumMaxCapacity:= 0;

// Loop over all childs
FOR ii:=0 TO usiNumOfLines-1 BY 1 DO
	// Build sum of all lines		
	dinSumMaxCapacity:= dinSumMaxCapacity + a_pLineChildSIF[ii]^.Cur.dinMaxCapacity; 	
END_FOR

// Return result
CalcMaxCapacity:= dinSumMaxCapacity;
END_METHOD

METHOD PROTECTED CalcSumOfItems : DINT
VAR
	ii: INT;
	dinSumOfItems: DINT;
END_VAR
// Method calculate the sum of hangers from all lines and return the result.

//Init
CalcSumOfItems:= 0;
dinSumOfItems:= 0;

// Loop over all childs
FOR ii:=0 TO usiNumOfLines-1 BY 1 DO
	// Build sum of all zones		
	dinSumOfItems:= dinSumOfItems + a_pLineChildSIF[ii]^.Cur.dinNumOfHangersInBuffer; 	
END_FOR

// Return result
CalcSumOfItems:= dinSumOfItems;
END_METHOD

METHOD checkChildAlmClass : BOOL
//------------------------------------------------------------------------------------------------------
// check child alarm classes
// set me alarm class active if at least one child has an EOFF
IF CheckAllChildAlmClass(E_AlmClass.EOFF) THEN
	CIf.Job.eMe_ActivAlmClass := E_AlmClass.EOFF;
	me.Alarm.bolfp := TRUE;
ELSIF CheckAllChildAlmClass(E_AlmClass.OFF) THEN
	CIf.Job.eMe_ActivAlmClass := E_AlmClass.OFF;
	me.Alarm.bolfp := TRUE;
ELSIF CheckAllChildAlmClass(E_AlmClass.STOP) THEN  // FB_MER needs alarm class STOP
	CIf.Job.eMe_ActivAlmClass := E_AlmClass.STOP;
	me.Alarm.bolfp := TRUE;
ELSE
	IF (me.Alarm.bolfp) THEN
		CIf.Job.eMe_ActivAlmClass := E_AlmClass.NONE; // no reset necessary
		me.Alarm.bolfp := FALSE;
	END_IF
END_IF

//------------------------------------------------------------------------------------------------------
// set alarm class parent of childs
//------------------------------------------------------------------------------------------------------
// set alarm class parent of childs in the case of a parent EOFF or me=OFF or EOFF
IF (CIf.Job.eParent_ActivAlmClass=E_AlmClass.EOFF) THEN
	SetAllChildAlmClass(CIf.Job.eParent_ActivAlmClass);
ELSIF(CIf.Job.eMe_ActivAlmClass=E_AlmClass.EOFF) OR (CIf.Job.eMe_ActivAlmClass=E_AlmClass.OFF) THEN
	SetAllChildAlmClass(CIf.Job.eMe_ActivAlmClass);
ELSE
	// no important alarm for child active
	SetAllChildAlmClass(E_AlmClass.NONE);
END_IF
END_METHOD

METHOD PROTECTED checkChildValid : BOOL
IF (usiNumOfLines = usiNumOfValidPointerToLine) THEN
	checkChildValid:= TRUE;
ELSE
	checkChildValid:= FALSE;
	// Invalid child pointer
	IF (usiNumOfLines <> usiNumOfValidPointerToLine) THEN
		// SIf.Alm[1].strText := 'Invalid child pointer'; 
		pfbAlarmCtrl^.setAlarm(CIf.Info.intCtrlId,1,0,ADR(SIf.Alm),E_AlmState.RST,CIf.Job.eMe_ActivAlmClass);	
	END_IF
END_IF
END_METHOD

METHOD PROTECTED checkStateAllLines : BOOL
VAR_INPUT
	cSTA: INT;
END_VAR
VAR
	ii: INT;
	usiNumOfCheckedChilds: USINT;
END_VAR
// Method check input state of all lines

//Init
checkStateAllLines:= FALSE;
usiNumOfCheckedChilds:= 0;

// Loop over all childs
FOR ii:=0 TO usiNumOfLines-1 BY 1 DO
	// Check state	
	// Special condition: In case if the child is in state ERROR and STOP is requested. Set child as checked.
	// Parent controller need state STOP that automatic stop sequence can work for all other childs.
	IF (a_pLineChildCIF[ii]^.Job.intState = cSTA) OR ((a_pLineChildCIF[ii]^.Job.intState = cSTA_ERROR) AND (cSTA = cSTA_STOP)) THEN
		usiNumOfCheckedChilds:= usiNumOfCheckedChilds+1;
		SIf.Cur.a_bolChildReady[ii] := TRUE;
	ELSE
		SIf.Cur.a_bolChildReady[ii] := FALSE;		
	END_IF

END_FOR

// All states equal the input state
IF (usiNumOfCheckedChilds = usiNumOfLines) THEN
	checkStateAllLines:= TRUE;
END_IF
END_METHOD

METHOD PROTECTED CmdToAllLines
VAR_INPUT
	cCMD: INT;
END_VAR
VAR
	ii: INT;
END_VAR
// Method send input command to all existing line child controller.
FOR ii:=0 TO usiNumOfLines-1 BY 1 DO	
	a_pLineChildCIF[ii]^.Job.intACmd:= cCMD;
END_FOR
END_METHOD

METHOD PROTECTED CtrlInit : BOOL
VAR
	ii: INT;
END_VAR
SUPER^.CtrlInit();

//----------------------------------------------------------------------
// Initialize all lines
//----------------------------------------------------------------------

// Method initialize all line child controller.
FOR ii:=0 TO usiNumOfLines-1 BY 1 DO	
	a_pLineChildCIF[ii] := THIS^.AddChild(a_pLineChildCtrl[ii]^);
	a_pLineChildSIF[ii] := a_pLineChildCtrl[ii]^.getCtrlSIf();
END_FOR

//----------------------------------------------------------------------
// Check about invalid configuration
//----------------------------------------------------------------------

// Check about invalid configuration of "MergeIntoTrp" mode. If one line is configured with this mode, set all other lines to the same mode.
bolModeMergeIntoTrpUsed:= FALSE;
// Check if any line is configured with "MergeIntoTrp" mode.
FOR ii:= 0 TO (usiNumOfLines-1) DO
	IF (SIf.Par.a_LinePar[ii].usiMergeMode = E_Typ_MER_AUTO_MODE.MergeIntoTrp) THEN
		// Mode is used
		bolModeMergeIntoTrpUsed:= TRUE;
		EXIT;
	END_IF
END_FOR
// Set  all other lines to "MergeIntoTrp" mode.
IF (bolModeMergeIntoTrpUsed = TRUE) THEN
	FOR ii:= 0 TO (usiNumOfLines-1) DO
		SIf.Par.a_LinePar[ii].usiMergeMode:= E_Typ_MER_AUTO_MODE.MergeIntoTrp;
	END_FOR	
END_IF

//----------------------------------------------------------------------
// Determine position of the last line
//----------------------------------------------------------------------
dinPositionOfLastLine_um:= SIf.Par.a_LinePar[usiNumOfLines-1].dinLinePosition_um;
END_METHOD

METHOD FB_init : BOOL
VAR_INPUT
	///if TRUE, the retain variables are initialized (warm start / cold start)
	bInitRetains: BOOL;
	///if TRUE, the instance afterwards gets moved into the copy code (online change)
	bInCopyCode: BOOL;
END_VAR
VAR
	ii: UINT;
END_VAR
//------------------------------------------------------------------------------------------------------------------------
// to manually change in new FUB implementation!!!
// define valid commands for this controller
FOR ii:= 0 TO (SIZEOF(CIf.Job.aCmdList)/SIZEOF(CIf.Job.aCmdList[0])-1) BY 1 DO
	IF (CIf.Job.aCmdList[ii].intCmd=cCMD_INITIALIZED) THEN
		// found first empty array element
		EXIT;
	END_IF
END_FOR

CIf.Job.aCmdList[ii].intCmd := cCMD_STOP;
CIf.Job.aCmdList[ii].strName := 'Stop'; 
CIf.Job.aCmdList[ii].bolAvailable := TRUE;
ii := ii +1;
CIf.Job.aCmdList[ii].intCmd := cCMD_RUN;
CIf.Job.aCmdList[ii].strName := 'Run';
CIf.Job.aCmdList[ii].bolAvailable := TRUE;

// set name of class/typ
CIf.Info.strType := 'FB_MER'; 

// set alarm class
SIf.Alm[1].eAlmClass := E_AlmClass.STOP;
SIf.Alm[1].strText := 'Invalid child pointer';
SIf.Alm[2].eAlmClass := E_AlmClass.INFO;
SIf.Alm[2].strText := 'Invalid line number. Line not exist';
SIf.Alm[3].eAlmClass := E_AlmClass.INFO;
SIf.Alm[3].strText := 'Merger waits for jam sensor free'; 


//*******************************************************************************
// initial values
//*******************************************************************************

// software configuration
CIf.SwCfg.bolExist := TRUE;
CIf.SwCfg.bolSimulation := FALSE;

// configuration
SIf.Cfg.usiMergeMainMode:= E_Typ_MER_MODE.Automatic;
SIf.Cfg.usiCountJamSensors:= 0;

// parameter
SIf.Par.udi_jamTimeout_ms:= 500;
// Default parameter for the lines are set in method InitLines
END_METHOD

METHOD PROTECTED getCmdState : STRING
VAR_INPUT
	intCmdState: INT;
	bolState: BOOL;
END_VAR
getCmdState := SUPER^.getCmdState(intCmdState:=intCmdState,bolState:=bolState); // get global/base defined cmds/states
IF (getCmdState='') THEN // global not defined get local
	// get string cmd/state string information in runtime
	IF (bolState=FALSE) THEN
		// cmd's
		CASE intCmdState OF
		END_CASE;
	ELSE
	
	// states
		CASE intCmdState OF	
			// SUB States
			cSTA_SUB_INITIALIZED:
				getCmdState := 'cSTA_SUB_INITIALIZED';			
			cSTA_SUB_WAIT_FOR_CMD:
				getCmdState := 'cSTA_SUB_WAIT_FOR_CMD';					
			cSTA_SUB_CHECK_HANGER_EXIST:
				getCmdState := 'cSTA_SUB_CHECK_HANGER_EXIST';
			cSTA_SUB_SEND_RELEASE:
				getCmdState := 'cSTA_SUB_SEND_RELEASE';
			cSTA_SUB_SEND_RELEASE_ALL:
				getCmdState := 'cSTA_SUB_SEND_RELEASE_ALL';	
			cSTA_SUB_SEND_STOP:
				getCmdState := 'cSTA_SUB_SEND_STOP';		
			cSTA_SUB_WAIT_JOB_DONE:
				getCmdState := 'cSTA_SUB_WAIT_JOB_DONE';
			cSTA_SUB_CHECK_MERGE_CON:
				getCmdState := 'cSTA_SUB_CHECK_MERGE_CON';
			cSTA_SUB_WAIT_LINE_FREE:
				getCmdState := 'cSTA_SUB_WAIT_LINE_FREE';	
			cSTA_SUB_END:
				getCmdState := 'cSTA_SUB_END';	
		END_CASE;
	END_IF
END_IF
END_METHOD

METHOD getCtrlSIf : POINTER TO T_Ctrl_SIf_MER
getCtrlSIf := ADR(SIf);
END_METHOD

METHOD PROTECTED IoInBridge : BOOL
// digitale and analoge inputs read from hardware or forcing
SIf.In.bolHangerDetected.map := THIS^.In_bolHangerDetected;
SIf.In.bolPinDetected.map := THIS^.In_bolPinDetected;

// Read sensors for waiting if a jam is detected
FOR intI := 1 TO SIf.Cfg.usiCountJamSensors DO
	SIf.In.a_bolJamSensor[intI].map := THIS^.In_a_bolJamSensor[intI];
	IF (CIf.SwCfg.bolSimulation = FALSE) THEN
		getInBol(CIf.Job.bolIoForce,ADR(SIf.In.a_bolJamSensor[intI]));
	END_IF
END_FOR

IF (CIf.SwCfg.bolSimulation = FALSE) THEN
	getInBol(CIf.Job.bolIoForce,ADR(SIf.In.bolHangerDetected));
	getInBol(CIf.Job.bolIoForce,ADR(SIf.In.bolPinDetected));
	//ctrl.In.bol_PosSwitchBasicDefTyp.intern := getInBol(ctrl.ifc.Job.bol_Force ,ADR(ctrl.In.bol_PosSwitchBasicDefTyp);
ELSE
	//simulation of global IO
END_IF
END_METHOD

METHOD PROTECTED IoOutBridge : BOOL
// digitale and analoge inputs read from hardware or forcing

// ... no physical outputs

IF (CIf.SwCfg.bolSimulation = FALSE) THEN
	// check interlocks to prevent damages
	IF (CIf.Job.bolIlkOverwrite=FALSE) THEN
		;
	END_IF
END_IF
END_METHOD

PROPERTY MaxCapacity : DINT
GET
MaxCapacity:= SIf.Cur.dinMaxCapacity;
END_GET
END_PROPERTY

PROPERTY NumOfHangers : DINT
GET
NumOfHangers:= SIf.Cur.dinCurrentItemCount;
END_GET
END_PROPERTY

METHOD PROTECTED sta_OFF : BOOL
// state implemetation
//--------------------------------------------------------------------------------------
// Entry action
	IF (me.StateMachine.intState<>me.StateMachine.intStateLastCycle) THEN
		me.StateMachine.intStateLastCycle := me.StateMachine.intState;
		;		
	END_IF

//--------------------------------------------------------------------------------------
// Cyclic action
	IF (me.StateMachine.intState=me.StateMachine.intStateLastCycle) THEN
		
		// Reset total counter
		SIf.Cur.dinNumOfMergedHangersTotal:= 0;
		
		// State Change Condition
		IF (me.Alarm.eActivAlmClass<>E_AlmClass.EOFF) AND (me.Alarm.eActivAlmClass<>E_AlmClass.OFF) THEN
			IF (me.intCmd=cCMD_STOP) THEN
				me.StateMachine.intStateNext := cSTA_STOPBusy;
			ELSIF (me.intCmd=cCMD_RUN) THEN 
				me.StateMachine.intStateNext := cSTA_RUNBusy;
			END_IF
		END_IF
	END_IF

//--------------------------------------------------------------------------------------
// Exit action
	IF (me.StateMachine.intState<>me.StateMachine.intStateNext) THEN
		;
	END_IF
END_METHOD

METHOD PROTECTED sta_RUN : BOOL
VAR
	/// Looping variable
	intSec: INT;
END_VAR
// state implemetation
//--------------------------------------------------------------------------------------
// Entry action
	IF (me.StateMachine.intState<>me.StateMachine.intStateLastCycle) THEN
		me.StateMachine.intStateLastCycle := me.StateMachine.intState;	
		;	
	END_IF

//--------------------------------------------------------------------------------------
// Cyclic action
	IF (me.StateMachine.intState=me.StateMachine.intStateLastCycle) THEN
			
		//-------------------------------------------------
		// Handling to merge into a transport belt
		//-------------------------------------------------	
		
		// Check if mode "MergeIntoTrp" is configured. 
		// If one line is configured with this mode, all other lines will be set to the same mode automatically in CtrlInit. Mixed mode not possible.
		IF ((SIf.Cfg.usiMergeMainMode = E_Typ_MER_MODE.Automatic) AND (SIf.Par.a_LinePar[0].usiMergeMode = E_Typ_MER_AUTO_MODE.MergeIntoTrp)) THEN
						
			//----------------------------------------------------------------------
			// Set the section start and end positions (triggered by pin sensor)
			//----------------------------------------------------------------------
			
			// Simulation of section start and end
			IF (CIf.SwCfg.bolSimulation = TRUE) THEN		
				SIf.In.bolPinDetected.intern:= FALSE;
				
				IF (dinSimWayTrigSection_um >= dinSimSectionLength_um) THEN
					dinSimWayTrigSection_um:= 0;
					// Set true for one cycle
					SIf.In.bolPinDetected.intern:= TRUE;
				END_IF
				// Increase position		
				dinSimWayTrigSection_um:= dinSimWayTrigSection_um + dinDrivenWay_um;
			END_IF
					
			// Wait for positive edge of the pin sensor (pin detected)
			IF (SIf.In.bolPinDetected.intern = TRUE) AND (bolRE_PinDetected = FALSE) THEN
				bolRE_PinDetected := TRUE;
					
				// Loop over section buffer
				FOR intSec := 0 TO cusiSectionBuffer_SIZE DO
					
					// If start position already set
					IF (a_stSectionBuffer[intSec].usiState = 1) THEN						
						// Set end position of the section
						a_stSectionBuffer[intSec].dinSecEndPos:= 0 - SIf.Par.dinPinLenght_um;
						a_stSectionBuffer[intSec].usiState:= 2;
					END_IF
					
					// Free buffer element  
					IF (a_stSectionBuffer[intSec].usiState = 0) THEN			
						// Set start position of the section
						a_stSectionBuffer[intSec].dinSecStartPos:= 0 - SIf.Par.dinPinLenght_um;
						a_stSectionBuffer[intSec].usiState:= 1;
						EXIT;									  
					END_IF
													
				END_FOR
					
			ELSIF (SIf.In.bolPinDetected.intern = FALSE) AND (bolRE_PinDetected = TRUE) THEN
				bolRE_PinDetected := FALSE;
			END_IF
			
			//----------------------------------------------------------------------
			// Set section engaged (hanger in section)
			//----------------------------------------------------------------------
			
			// Wait for positive edge of the hanger sensor
			IF (SIf.In.bolHangerDetected.intern = TRUE) AND (bolRE_HangerDetected = FALSE) THEN
				bolRE_HangerDetected := TRUE;
					
				// Loop over section buffer to mark buffer element with 3 = section engaged (hanger in section detected by hanger sensor)
				FOR intSec := 0 TO cusiSectionBuffer_SIZE-1 DO		
					
					// Prio 1: Normal sequence.
					IF (SIf.Par.dinHangerSensorPosition_um < a_stSectionBuffer[intSec].dinSecStartPos) AND  
						(SIf.Par.dinHangerSensorPosition_um > (a_stSectionBuffer[intSec].dinSecEndPos - SIf.Par.dinPinLenght_um)) THEN	
							// Mark the buffer element with 3 = section engaged (hanger in section detected by hanger sensor)
							a_stSectionBuffer[intSec].usiState:= 3;
						EXIT;
					
					// Prio 2: If range is not accurately recognized mark buffer element X and X +1.
					ELSIF (SIf.Par.dinHangerSensorPosition_um < a_stSectionBuffer[intSec].dinSecEndPos) AND  
						(SIf.Par.dinHangerSensorPosition_um > a_stSectionBuffer[intSec+1].dinSecStartPos) THEN	
							// Mark the buffer element with 3 = section engaged (hanger in section detected by hanger sensor)
							a_stSectionBuffer[intSec].usiState:= 3;
							a_stSectionBuffer[intSec+1].usiState:= 3;
						EXIT;
					END_IF		
						
				END_FOR	
					
			ELSIF (SIf.In.bolHangerDetected.intern = FALSE) AND (bolRE_HangerDetected = TRUE) THEN
				bolRE_HangerDetected := FALSE;
			END_IF	
				
			//----------------------------------------------------------------------
			// Buffer tracking 
			//----------------------------------------------------------------------
			
			// Move all buffer elements 1 down if hanger was released. State will be set to "0" in state RUN if a hanger is released.
			// Also check if a section is driven out!			
			IF (a_stSectionBuffer[0].usiState = 0) OR (a_stSectionBuffer[0].dinSecEndPos > (dinPositionOfLastLine_um + SIf.Par.dinSectionLenght_um))THEN
				// Loop every buffer element 1 Down
				FOR intSec := 0 TO cusiSectionBuffer_SIZE-1 DO			
					a_stSectionBuffer[intSec].dinSecStartPos := a_stSectionBuffer[intSec+1].dinSecStartPos;
					a_stSectionBuffer[intSec].dinSecEndPos := a_stSectionBuffer[intSec+1].dinSecEndPos;
					a_stSectionBuffer[intSec].dinTrigStartPos := a_stSectionBuffer[intSec+1].dinTrigStartPos;
					a_stSectionBuffer[intSec].dinTrigEndPos := a_stSectionBuffer[intSec+1].dinTrigEndPos;
					a_stSectionBuffer[intSec].usiState := a_stSectionBuffer[intSec+1].usiState;
				END_FOR		
				a_stSectionBuffer[intSec].dinSecStartPos := 0;
				a_stSectionBuffer[intSec].dinSecEndPos := 0;
				a_stSectionBuffer[intSec].dinTrigStartPos := 0;
				a_stSectionBuffer[intSec].dinTrigEndPos := 0;
				a_stSectionBuffer[intSec].usiState := 0;
			END_IF
			
			//----------------------------------------------------------------------
			// Increase positions
			//----------------------------------------------------------------------
				
			// Increase the buffer positions
			FOR intSec := 0 TO cusiSectionBuffer_SIZE DO
				
				IF (a_stSectionBuffer[intSec].usiState = 1) THEN
					// Section start/end
					a_stSectionBuffer[intSec].dinSecStartPos:= a_stSectionBuffer[intSec].dinSecStartPos + dinDrivenWay_um;
					// Trigger start/end
					a_stSectionBuffer[intSec].dinTrigStartPos:= a_stSectionBuffer[intSec].dinSecStartPos - SIf.Par.dinTrigStartOffset_um;
					a_stSectionBuffer[intSec].dinTrigEndPos:= a_stSectionBuffer[intSec].dinSecStartPos - SIf.Par.dinTrigEndOffset_um;	
					
				ELSIF (a_stSectionBuffer[intSec].usiState >= 2) THEN
					// Section start/end
					a_stSectionBuffer[intSec].dinSecStartPos:= a_stSectionBuffer[intSec].dinSecStartPos + dinDrivenWay_um;
					a_stSectionBuffer[intSec].dinSecEndPos:= a_stSectionBuffer[intSec].dinSecEndPos + dinDrivenWay_um;
					// Trigger start/end
					a_stSectionBuffer[intSec].dinTrigStartPos:= a_stSectionBuffer[intSec].dinSecStartPos - SIf.Par.dinTrigStartOffset_um;
					a_stSectionBuffer[intSec].dinTrigEndPos:= a_stSectionBuffer[intSec].dinSecStartPos - SIf.Par.dinTrigEndOffset_um;				
				END_IF
				
			END_FOR	
			
		END_IF
	
		
		// Check States for parent information
		THIS^.checkStateAllLines(cSTA_RUN);

		// Check jam detection
		IF (udiJamReleaseDelayTime_ms > SIf.Par.udi_jamTimeout_ms) THEN
			bolJamDetected := FALSE;
		ELSE
			udiJamReleaseDelayTime_ms := udiJamReleaseDelayTime_ms + me.FUBInfo.udiSample_ms;
		END_IF
		
		FOR intI := 1 TO SIf.Cfg.usiCountJamSensors DO
			// Start jam timer
			IF ((SIf.In.a_bolJamSensor[intI].intern = TRUE) AND (a_bolJamSensorOnce[intI] = FALSE)) THEN
				a_bolJamSensorOnce[intI]:= TRUE;
				//a_udiTimeJamDetection[intI]:= me.StateMachine.udiTimeInState_ms;
				a_udiTimeJamDetection[intI]:= 0;
			// Stop jam timer
			ELSIF ((SIf.In.a_bolJamSensor[intI].intern = FALSE) AND (a_bolJamSensorOnce[intI] = TRUE)) THEN
				a_bolJamSensorOnce[intI]:= FALSE;
			// Set flag if neccessary
			ELSIF ((SIf.In.a_bolJamSensor[intI].intern = TRUE) AND (a_bolJamSensorOnce[intI] = TRUE)) THEN
				//IF (me.StateMachine.udiTimeInState_ms > a_udiTimeJamDetection[intI] + SIf.Par.udi_jamTimeout_ms) THEN
				IF (a_udiTimeJamDetection[intI] > SIf.Par.udi_jamTimeout_ms) THEN
					bolJamDetected := TRUE;
					udiJamReleaseDelayTime_ms := 0;
				END_IF
			END_IF
			a_udiTimeJamDetection[intI]:= a_udiTimeJamDetection[intI]+ me.FUBInfo.udiSample_ms;
		END_FOR
	
		//----------------------------------------------------------------------------------------
		// Substates for merging lines dependent time or distribution of the number of hangers
		//----------------------------------------------------------------------------------------
		CASE me.SubStateMachine.intState OF
	
			//-----------------------------------------------
			// INITIALIZE 					(MODE: All modes)
			//-----------------------------------------------
			cSTA_SUB_INITIALIZED:
			
				// Check configured main mode
				CASE SIf.Cfg.usiMergeMainMode OF	
				
					// Mode - Automatic
					E_Typ_MER_MODE.Automatic:		
						me.SubStateMachine.intStateNext := cSTA_SUB_CHECK_HANGER_EXIST;					
									
					// Mode - OnCommand	
					E_Typ_MER_MODE.OnCommand:		
						me.SubStateMachine.intStateNext := cSTA_SUB_WAIT_FOR_CMD;
														
				END_CASE
			
			//-----------------------------------------------
			// WAIT FOR COMMAND 			(MODE: OnCommand)
			//-----------------------------------------------	
			cSTA_SUB_WAIT_FOR_CMD:
			
				// Wait for command to release all
				IF (me.intCmd=SLB_CmdState.cCMD_RELEASE_ALL) THEN
					// Check about valid line number
					IF ((SIf.Par.usiLineNumToReleaseAll = 0) OR (SIf.Par.usiLineNumToReleaseAll > usiNumOfLines)) THEN
						// Invalid line	
						// SIf.Alm[2].strText := 'Invalid line number. Line not exist'; 
						pfbAlarmCtrl^.setAlarm(CIf.Info.intCtrlId,2,0,ADR(SIf.Alm),E_AlmState.RST,CIf.Job.eMe_ActivAlmClass);		
					ELSE
						// Valid line	
						usiLineNumToReleaseAll:= SIf.Par.usiLineNumToReleaseAll-1;
						me.SubStateMachine.intStateNext := cSTA_SUB_SEND_RELEASE_ALL;
					END_IF
						
				END_IF
				
			//-----------------------------------------------
			// CHECK HANGER EXIST 			(MODE: Automatic)     
			//-----------------------------------------------
			cSTA_SUB_CHECK_HANGER_EXIST:
				// Entry action
				IF (me.SubStateMachine.intState<>me.SubStateMachine.intStateLastCycle) THEN
					me.SubStateMachine.intStateLastCycle := me.SubStateMachine.intState;							
					;						
				END_IF
		
				// Init
				bolReleaseHanger:= FALSE;
				bolSectionFree := FALSE;
						
				// Check if mode "MergeIntoTrp" is configured.
				IF (SIf.Par.a_LinePar[usiIndexToRelease].usiMergeMode = E_Typ_MER_AUTO_MODE.MergeIntoTrp) THEN
					FOR intSec := 0 TO cusiSectionBuffer_SIZE DO
						// Check if the current line position is within the trigger window to release the hanger
						IF ((SIf.Par.a_LinePar[usiIndexToRelease].dinLinePosition_um < a_stSectionBuffer[intSec].dinTrigStartPos)
							AND (SIf.Par.a_LinePar[usiIndexToRelease].dinLinePosition_um > a_stSectionBuffer[intSec].dinTrigEndPos)
							AND (a_stSectionBuffer[intSec].usiState = 2)) THEN
								// Section is free, hanger can be released
								bolSectionFree := TRUE;	
								EXIT;
						END_IF
					END_FOR					
				END_IF
					
				// Check hanger exists on line
				IF (((a_pLineChildSIF[usiIndexToRelease]^.Cur.bolHangerDetected=TRUE) AND (SIf.Par.a_LinePar[usiIndexToRelease].usiMergeMode <> E_Typ_MER_AUTO_MODE.MergeIntoTrp)) OR
					((a_pLineChildSIF[usiIndexToRelease]^.Cur.bolHangerDetected=TRUE) AND (bolSectionFree = TRUE) AND (SIf.Par.a_LinePar[usiIndexToRelease].usiMergeMode = E_Typ_MER_AUTO_MODE.MergeIntoTrp))) THEN		

					IF (SIf.Par.a_LinePar[usiIndexToRelease].usiMergeMode = E_Typ_MER_AUTO_MODE.MergeIntoTrp) THEN
						// Mark the buffer element with 4 = hanger released (section engaged)
						a_stSectionBuffer[intSec].usiState:= 4;	
					END_IF
					bolReleaseHanger:= TRUE;
					
				ELSE		
					// No hanger on this line, check next
					IF (usiIndexToRelease < (usiNumOfLines-1)) THEN
						// Inc. index to next line
						usiIndexToRelease:= usiIndexToRelease + 1;	
					ELSE
						usiIndexToRelease:= 0;
					END_IF
				END_IF			

		
				// State Change Condition
				IF (bolReleaseHanger=TRUE) THEN
					me.SubStateMachine.intStateNext := cSTA_SUB_SEND_RELEASE;
					// Reset counter and timer
					dinNumOfPassedHangers:=0;
					udiMergingTime:=0;
				END_IF
						
			//-----------------------------------------------
			// SEND RELEASE					(MODE: Automatic)
			//-----------------------------------------------
			cSTA_SUB_SEND_RELEASE:		
	
				// Send release command to line X (trigger command)
				a_pLineChildCIF[usiIndexToRelease]^.Job.intACmd:= STB_CmdState.cCMD_RELEASE;				
				
				// State Change Condition
				IF(TRUE)THEN
					me.SubStateMachine.intStateNext := cSTA_SUB_WAIT_JOB_DONE;					
				END_IF	
						
			//-----------------------------------------------
			// SEND RELEASE	ALL				(MODE: OnCommand)
			//-----------------------------------------------
			cSTA_SUB_SEND_RELEASE_ALL:
			
				// Send release all command to line X
				a_pLineChildCIF[usiLineNumToReleaseAll]^.Job.intACmd:= STB_CmdState.cCMD_RELEASE_ALL;				
				
				// State Change Condition
				IF(TRUE)THEN
					me.SubStateMachine.intStateNext := cSTA_SUB_WAIT_JOB_DONE;					
				END_IF		
					
			//-----------------------------------------------
			// WAIT JOB DONE				(MODE: All modes)
			//-----------------------------------------------
			cSTA_SUB_WAIT_JOB_DONE:
		
				// Check configured main mode
				CASE SIf.Cfg.usiMergeMainMode OF	
				
					// Mode - Automatic
					E_Typ_MER_MODE.Automatic:
						// State Change Condition
						// Wait until job done
						IF(a_pLineChildCIF[usiIndexToRelease]^.Job.intACmd = cSTA_DONE)THEN									
							IF (SIf.Par.a_LinePar[usiIndexToRelease].usiMergeMode = E_Typ_MER_AUTO_MODE.MergeIntoTrp) THEN							
								me.SubStateMachine.intStateNext := cSTA_SUB_WAIT_LINE_FREE;							
							ELSE
								me.SubStateMachine.intStateNext := cSTA_SUB_CHECK_MERGE_CON;
							END_IF																					
						END_IF	
									
					// Mode - OnCommand	
					E_Typ_MER_MODE.OnCommand:
						// State Change Condition
						// Wait until release all
						IF(a_pLineChildCIF[usiLineNumToReleaseAll]^.Job.intState = SLB_CmdState.cCMD_RELEASE_ALL)THEN				
							me.SubStateMachine.intStateNext := cSTA_SUB_SEND_STOP;																
						END_IF
						
				END_CASE
							
			//-----------------------------------------------
			// SEND STOP					(MODE: OnCommand)
			//-----------------------------------------------
			cSTA_SUB_SEND_STOP:
			
				// Send stop command to line X
				a_pLineChildCIF[usiLineNumToReleaseAll]^.Job.intACmd:=cCMD_RUN;				
				
				// State Change Condition
				IF(a_pLineChildCIF[usiLineNumToReleaseAll]^.Job.intState=cSTA_RUN)THEN
					me.SubStateMachine.intStateNext := cSTA_SUB_WAIT_LINE_FREE;					
				END_IF	
								
			//-----------------------------------------------
			// CHECK MERGE CONDITIONS		(MODE: Automatic)
			//-----------------------------------------------
			cSTA_SUB_CHECK_MERGE_CON:
				// Entry action
				IF (me.SubStateMachine.intState<>me.SubStateMachine.intStateLastCycle) THEN
					me.SubStateMachine.intStateLastCycle := me.SubStateMachine.intState;							
					;						
				END_IF
					
				// Count the passed hangers from current line X
				IF (a_pLineChildSIF[usiIndexToRelease]^.Cur.dinHangersPassedTotal <> dinPassedTotalLineXOld) THEN
					// Count passed hangers if "E_Typ_MER_AUTO_MODE.MergeOverSetpoint" is selected.				
					dinNumOfPassedHangers:= dinNumOfPassedHangers + a_pLineChildSIF[usiIndexToRelease]^.Cur.uinNumOfHangersPerPulseFirstZone;			
					// Calculate merged hangers total
					SIf.Cur.dinNumOfMergedHangersTotal:= SIf.Cur.dinNumOfMergedHangersTotal + a_pLineChildSIF[usiIndexToRelease]^.Cur.uinNumOfHangersPerPulseFirstZone;									
				END_IF
				dinPassedTotalLineXOld:= a_pLineChildSIF[usiIndexToRelease]^.Cur.dinHangersPassedTotal;
		
					
				// State Change Condition
				IF (a_pLineChildSIF[usiIndexToRelease]^.Cur.bolHangerDetected=FALSE) THEN	// No hanger exist
					me.SubStateMachine.intStateNext := cSTA_SUB_WAIT_LINE_FREE;				
				ELSIF ((SIf.Par.a_LinePar[usiIndexToRelease].usiMergeMode = E_Typ_MER_AUTO_MODE.MergeOverTime) AND (udiMergingTime >= SIf.Par.a_LinePar[usiIndexToRelease].udiMergingTime_ms)) THEN
					me.SubStateMachine.intStateNext := cSTA_SUB_WAIT_LINE_FREE;				
				ELSIF ((SIf.Par.a_LinePar[usiIndexToRelease].usiMergeMode = E_Typ_MER_AUTO_MODE.MergeOverSetpoint) AND (dinNumOfPassedHangers >= SIf.Par.a_LinePar[usiIndexToRelease].uinNumOfHangersToMerge)) THEN
					me.SubStateMachine.intStateNext := cSTA_SUB_WAIT_LINE_FREE;							
				ELSIF ((SIf.Par.a_LinePar[usiIndexToRelease].usiMergeMode = E_Typ_MER_AUTO_MODE.MergeOverTime) AND (udiMergingTime < SIf.Par.a_LinePar[usiIndexToRelease].udiMergingTime_ms)) THEN
					me.SubStateMachine.intStateNext := cSTA_SUB_SEND_RELEASE;					
				ELSIF ((SIf.Par.a_LinePar[usiIndexToRelease].usiMergeMode = E_Typ_MER_AUTO_MODE.MergeOverSetpoint) AND (dinNumOfPassedHangers < SIf.Par.a_LinePar[usiIndexToRelease].uinNumOfHangersToMerge)) THEN
					me.SubStateMachine.intStateNext := cSTA_SUB_SEND_RELEASE;	
				END_IF
	
			//-----------------------------------------------
			// WAIT UNTIL LINE IS FREE		(MODE: All modes)
			//-----------------------------------------------
			cSTA_SUB_WAIT_LINE_FREE:

				IF (bolJamDetected	= TRUE) THEN // Line is not free, jam detected
					// SIf.Alm[3].strText := 'Merger waits for jam sensor free';
					pfbAlarmCtrl^.setAlarm(CIf.Info.intCtrlId,3,0,ADR(SIf.Alm),E_AlmState.RST,CIf.Job.eMe_ActivAlmClass);				
				ELSE				
					// Check configured main mode
					CASE SIf.Cfg.usiMergeMainMode OF	
					
						// Mode - Automatic
						E_Typ_MER_MODE.Automatic:
							// State Change Condition
							IF (me.SubStateMachine.udiTimeInState_ms > SIf.Par.a_LinePar[usiIndexToRelease].udiWaitTimeLineFree_ms) OR 
								(SIf.Par.a_LinePar[usiIndexToRelease].usiMergeMode = E_Typ_MER_AUTO_MODE.MergeIntoTrp) THEN
								IF(me.intCmd=cCMD_STOP)THEN
									// Go to end
									me.SubStateMachine.intStateNext := cSTA_SUB_END;
								ELSE
									// Merging cycle line X complete
									IF (usiIndexToRelease < (usiNumOfLines-1)) THEN						
										// Inc. index to next line
										usiIndexToRelease:= usiIndexToRelease + 1;	
									ELSE
										usiIndexToRelease:= 0;
									END_IF
									
									// Go on with automatic cycle
									me.SubStateMachine.intStateNext := cSTA_SUB_CHECK_HANGER_EXIST;					
								END_IF		
							END_IF
									
						// Mode - OnCommand	
						E_Typ_MER_MODE.OnCommand:
							// State Change Condition
							IF (me.SubStateMachine.udiTimeInState_ms > SIf.Par.a_LinePar[usiLineNumToReleaseAll].udiWaitTimeLineFree_ms) THEN												
								// Update merged hangers total -> After release all, use passed package 
								SIf.Cur.dinNumOfMergedHangersTotal:= SIf.Cur.dinNumOfMergedHangersTotal + a_pLineChildSIF[usiLineNumToReleaseAll]^.Cur.dinHangersPassedPackage;			
								
								IF(me.intCmd=cCMD_STOP)THEN
									// Go to end
									me.SubStateMachine.intStateNext := cSTA_SUB_END;
								ELSE
									//Set "Job done" for parent
									CIf.Job.intACmd:=cSTA_DONE;
									me.SubStateMachine.intStateNext := cSTA_SUB_WAIT_FOR_CMD;
								END_IF								
							END_IF
							
					END_CASE
				END_IF
			//-----------------------------------------------
			// END							(MODE: All modes)
			//-----------------------------------------------
			cSTA_SUB_END:
			     // ... do nothing
		
		END_CASE

		// Timer handling for merging time
		udiMergingTime:= udiMergingTime + me.FUBInfo.udiSample_ms;
			
		// State Change Condition
		IF ((me.intCmd=cCMD_STOP) AND ((me.SubStateMachine.intState=cSTA_SUB_END) OR (me.SubStateMachine.intState=cSTA_SUB_CHECK_HANGER_EXIST) OR (me.SubStateMachine.intState=cSTA_SUB_WAIT_FOR_CMD) OR (me.SubStateMachine.intState=cSTA_SUB_WAIT_LINE_FREE))) THEN
			me.StateMachine.intStateNext := cSTA_STOPBusy;
		END_IF
	END_IF

//--------------------------------------------------------------------------------------
// Exit action
	IF (me.StateMachine.intState<>me.StateMachine.intStateNext) THEN
		;
	END_IF
END_METHOD

METHOD PROTECTED sta_RUNBusy : BOOL
VAR
	ii: INT;
END_VAR
// state implemetation
//--------------------------------------------------------------------------------------
// Entry action
	IF (me.StateMachine.intState<>me.StateMachine.intStateLastCycle) THEN
		me.StateMachine.intStateLastCycle := me.StateMachine.intState;
	
		bolGoToRun:= FALSE;
		usiIndexToRelease:= 0;
		
		// Initialize sub state machine
		me.SubStateMachine.intState:= cSTA_SUB_INITIALIZED; 
		me.SubStateMachine.intStateNext:= cSTA_SUB_INITIALIZED;
		
	END_IF

//--------------------------------------------------------------------------------------
// Cyclic action
	IF (me.StateMachine.intState=me.StateMachine.intStateLastCycle) THEN
			
		// Check if mode "MergeIntoTrp" is configured. 
		IF ((SIf.Cfg.usiMergeMainMode = E_Typ_MER_MODE.Automatic) AND (SIf.Par.a_LinePar[0].usiMergeMode = E_Typ_MER_AUTO_MODE.MergeIntoTrp)) THEN
			// Clear section buffer
			FOR ii := 0 TO cusiSectionBuffer_SIZE DO
				a_stSectionBuffer[ii].dinSecStartPos := 0;
				a_stSectionBuffer[ii].dinSecEndPos := 0;
				a_stSectionBuffer[ii].dinTrigStartPos := 0;
				a_stSectionBuffer[ii].dinTrigEndPos := 0;
				a_stSectionBuffer[ii].usiState := 0;				
			END_FOR
		END_IF
		
		// Check configured main mode
		CASE SIf.Cfg.usiMergeMainMode OF	
		
			// Mode - Automatic
			E_Typ_MER_MODE.Automatic:
			
				// send command RUN to all existing line child controller.
				THIS^.CmdToAllLines(cCMD_RUN);
				
				// State Change Condition
				// Check if all childs in "RUN", ready for release hanger 
				IF(THIS^.checkStateAllLines(cSTA_RUN))THEN
					bolGoToRun:= TRUE;			
				END_IF	
		
			// Mode - OnCommand	
			E_Typ_MER_MODE.OnCommand:
			
				// send command STOP to all existing line child controller.
				THIS^.CmdToAllLines(cCMD_RUN);
				
				// State Change Condition
				// Check if all childs stopped, ready for new command 
				IF(THIS^.checkStateAllLines(cSTA_RUN))THEN
					bolGoToRun:= TRUE;					
				END_IF	
			
		END_CASE

	
		// State Change Condition	
		IF (bolGoToRun=TRUE) THEN
			me.StateMachine.intStateNext := cSTA_RUN;		
		END_IF

	END_IF

//--------------------------------------------------------------------------------------
// Exit action
	IF (me.StateMachine.intState<>me.StateMachine.intStateNext) THEN
		;
	END_IF
END_METHOD

METHOD PROTECTED sta_STOP : BOOL
// state implemetation
//--------------------------------------------------------------------------------------
// Entry action
	IF (me.StateMachine.intState<>me.StateMachine.intStateLastCycle) THEN
		me.StateMachine.intStateLastCycle := me.StateMachine.intState;
		;
	END_IF

//--------------------------------------------------------------------------------------
// Cyclic action
	IF (me.StateMachine.intState=me.StateMachine.intStateLastCycle) THEN

		// State Change Condition	
		IF (me.intCmd = cCMD_RUN) THEN 
			me.StateMachine.intStateNext := cSTA_RUNBusy;
		END_IF
	END_IF

//-------------------------------------------------------------------------------------
// Exit action
	IF (me.StateMachine.intState<>me.StateMachine.intStateNext) THEN
		;
	END_IF
END_METHOD

METHOD PROTECTED sta_STOPBusy : BOOL
// state implemetation
//--------------------------------------------------------------------------------------
// Entry action
	IF (me.StateMachine.intState<>me.StateMachine.intStateLastCycle) THEN
		me.StateMachine.intStateLastCycle := me.StateMachine.intState;
		
		// send command STOP to all existing line child controller.
		THIS^.CmdToAllLines(cCMD_STOP);

	END_IF

//--------------------------------------------------------------------------------------
// Cyclic action
	IF (me.StateMachine.intState=me.StateMachine.intStateLastCycle) THEN
			
		// State Change Condition
		// Check if all STOPPED
		IF (THIS^.checkStateAllLines(cSTA_STOP)) THEN
			me.StateMachine.intStateNext := cSTA_STOP;
		END_IF
	END_IF

//--------------------------------------------------------------------------------------
// Exit action
	IF (me.StateMachine.intState<>me.StateMachine.intStateNext) THEN
		;
	END_IF
END_METHOD

METHOD PROTECTED StateMachine : BOOL
SUPER^.StateMachine();

// main statemachine of base controller
CASE me.StateMachine.intState OF
    cSTA_STOPBusy: 
        THIS^.sta_STOPBusy();
    cSTA_STOP: 
        THIS^.sta_STOP();
	cSTA_RUNBusy: 
        THIS^.sta_RUNBusy();
    cSTA_RUN: 
        THIS^.sta_RUN();				
END_CASE;
END_METHOD

END_FUNCTION_BLOCK

// POUs/Controller/Lvl2/HFE/FB_HFE
FUNCTION_BLOCK FB_HFE EXTENDS FB_CtrlBase
VAR_INPUT
	a_bolLDSNeedsHanger: ARRAY[0..cuintMaxStation] OF BOOL;
	p_fbTlpDrive: POINTER TO FB_DRV;
	///p_fbJunction : POINTER TO FB_JUN;
	p_fbSLB: POINTER TO FB_SLB;
END_VAR
VAR
	/// List of pointers to Childs of VLV
	a_pMultiChildCtrl: ARRAY[0..Base_Const.cMaxNrOfChilds] OF POINTER TO FB_VLV;
	/// List of childs common interface
	a_pMultiChildCIF: ARRAY[0..Base_Const.cMaxNrOfChilds] OF POINTER TO T_Ctrl_CIf;
	/// List of childs specific interface for additional parameters or cur
	a_pMultiChildSIF: ARRAY[0..Base_Const.cMaxNrOfChilds] OF POINTER TO Base_Elements.T_Ctrl_SIf_VLV;
	usiNumOfMultiChild: USINT;
	usiNumOfValidPointerMultiChild: USINT;
	/// Specific interface struct for public access
	SIf: T_Ctrl_SIf_HFE;
	/// Child controller
	pTlpDrive_CIf: POINTER TO T_Ctrl_CIf;
	///pJunction_CIf : POINTER TO T_Ctrl_CIf;
	pSLB_CIf: POINTER TO T_Ctrl_CIf;
	pSLB_SIf: POINTER TO T_Ctrl_SIf_SLB;
	intSubState: ARRAY[0..cuintMaxStation] OF INT;
	udiTimeInStateRefill_ms: ARRAY[0..cuintMaxStation] OF UDINT;
END_VAR
VAR CONSTANT
	/// sub States
	cSTA_SUB_WaitForJob: INT := 500;
	cSTA_SUB_WaitOpen: INT := 502;
	cSTA_SUB_Open: INT := 504;
	cSTA_SUB_WaitClose: INT := 506;
	cSTA_SUB_Close: INT := 508;
END_VAR

(*__________________________________________________________________________________________________
¦	
¦	Vistaprint Schweiz GmbH
¦	CH - 8401 Winterthur
¦
¦	www.vistaprint.ch - info@vistaprint.ch
¦___________________________________________________________________________________________________

Function desription:
Cylinder implementation. 


History:
Version		Date			Author		Comment
---------------------------------------------------------------------------------------------------
0.00.1		02.07.2013		VP/RE		Start history
0.00.2		16.12.2013		AVME/MRU	In Always: No EOFF State!! in EOFF go to OFF

___________________________________________________________________________________________________*)



// check if child pointer valid
IF (me.bolActivate) AND (p_fbTlpDrive<>0)  AND (THIS^.checkChildPointer()) AND (p_fbSLB<>0) THEN // cyclic call enabled
	
	IF (CIf.Info.bolInitDone=FALSE) THEN // first cycle -> init
		CtrlInit();
		CIf.Info.bolInitDone := TRUE;
	ELSE
		CycleStartDuty();
	
		Always();
		
		StateMachine();
		
		CycleEndDuty();
	END_IF
	
END_IF;

METHOD AddJunction
VAR_INPUT
	p_MultiChild: POINTER TO FB_JUN;
END_VAR

// Method add the pointer address of the buffer zone child controller to the array list.
IF (usiNumOfMultiChild <= (Base_Const.cMaxNrOfChilds-1)) THEN
	// Add buffer zone child controller to list
	a_pMultiChildCtrl[usiNumOfMultiChild] := p_MultiChild;
	// Inc. number of buffer zones
	usiNumOfMultiChild:= usiNumOfMultiChild+1;
	// Check if the pointer is valid
	IF (p_MultiChild<>0) THEN
		usiNumOfValidPointerMultiChild:= usiNumOfValidPointerMultiChild+1;
	END_IF
END_IF
END_METHOD

METHOD PROTECTED Always : BOOL
SUPER^.Always();

IF (me.StateMachine.intState<>cSTA_SINGLE_ANSWER) THEN
	
	;
	
END_IF

// ----------------------------------------------------------------------------------
// Conditions Always
// overrule error always from base -> no EOFF State!! in EOFF go to OFF
IF (me.StateMachine.intStateNext = cSTA_EOFFBusy) THEN
	IF (me.StateMachine.intState=cSTA_OFF) THEN
		me.StateMachine.intStateNext := cSTA_OFF;
	ELSE // stay in OFF
		me.StateMachine.intStateNext := cSTA_OFFBusy;
	END_IF
END_IF
END_METHOD

METHOD PROTECTED checkChildPointer : BOOL
IF (usiNumOfMultiChild = usiNumOfValidPointerMultiChild) THEN
	checkChildPointer:= TRUE;
ELSE
	checkChildPointer:= FALSE;
END_IF
END_METHOD

METHOD PROTECTED CtrlInit : BOOL
VAR
	ii: INT;
END_VAR
SUPER^.CtrlInit();

// get child CIf
pTlpDrive_CIf := THIS^.AddChild(p_fbTlpDrive^);
pSLB_CIf := THIS^.AddChild(p_fbSLB^);
pSLB_SIf := p_fbSLB^.getCtrlSIf();

//initialize all multi Child controller.
FOR ii:=0 TO usiNumOfMultiChild-1 BY 1 DO	
	// Get child common if
	a_pMultiChildCIF[ii]:= THIS^.AddChild(a_pMultiChildCtrl[ii]^);	
	// Get specific interface for additional parmaeters or cur
	a_pMultiChildSIF[ii]:= a_pMultiChildCtrl[ii]^.getCtrlSIf();
END_FOR
END_METHOD

METHOD FB_init : BOOL
VAR_INPUT
	///if TRUE, the retain variables are initialized (warm start / cold start)
	bInitRetains: BOOL;
	///if TRUE, the instance afterwards gets moved into the copy code (online change)
	bInCopyCode: BOOL;
END_VAR
VAR
	ii: UINT;
END_VAR
//------------------------------------------------------------------------------------------------------------------------
// to manually change in new FUB implementation!!!
// define valid commands for this controller
FOR ii:= 0 TO (SIZEOF(CIf.Job.aCmdList)/SIZEOF(CIf.Job.aCmdList[0])-1) BY 1 DO
	IF (CIf.Job.aCmdList[ii].intCmd=cCMD_INITIALIZED) THEN
		// found first empty array element
		EXIT;
	END_IF
END_FOR
CIf.Job.aCmdList[ii].intCmd := cCMD_RUN;
CIf.Job.aCmdList[ii].strName := 'Run'; 
CIf.Job.aCmdList[ii].bolAvailable := TRUE;
//ii := ii +1;
//CIf.Job.aCmdList[ii].intCmd := cCMD_RETRACT;
//CIf.Job.aCmdList[ii].strName := 'Retract';
//CIf.Job.aCmdList[ii].bolAvailable := TRUE;

// set name of class/typ
CIf.Info.strType := 'FB_HFE'; 

// set alarm class
//SIf.Alm[1].eAlmClass := E_AlmClass.TSTOP;
//SIf.Alm[1].strText := 'TLKV Motor does not move after timeout.'; 
//SIf.Alm[2].eAlmClass := E_AlmClass.STOP;
//SIf.Alm[2].strText := 'Emergency button pressed.'; 

//*******************************************************************************
// initial values
//*******************************************************************************

// software configuration
CIf.SwCfg.bolExist := TRUE;
CIf.SwCfg.bolSimulation := FALSE;

// parmeter
SIf.Par.udiWaitingTime_ms := 100;
SIf.Par.a_bolEnableJunction[0] := TRUE; // First LDS is enabled

// configuration
SIf.Cfg.uintNbOfLDS := 1;

// actual values
//SIf.Cur.dinCounter := 0;
END_METHOD

METHOD getCtrlSIf : POINTER TO T_Ctrl_SIf_HFE
getCtrlSIf := ADR(SIf);
END_METHOD

METHOD PROTECTED IoInBridge : BOOL
// digitale and analoge inputs read from hardware or forcing
//SIf.In.bolGiveNextHangerSensor.map := THIS^.In_GiveNextHangerSensor;

IF (CIf.SwCfg.bolSimulation = FALSE) THEN
	//getInBol(CIf.Job.bolIoForce,ADR(SIf.In.bolGiveNextHangerSensor));
ELSE
	//simulation of global IO
END_IF
END_METHOD

METHOD PROTECTED IoOutBridge : BOOL
VAR
	bolSwitchValvesOff: BOOL;
END_VAR
// digitale and analoge inputs read from hardware or forcing
IF (CIf.SwCfg.bolSimulation = FALSE) THEN
	//setOutBol(CIf.Job.bolIoForce ,ADR(SIf.Out.bolClamping));

	//THIS^.Out_Clamping := SIf.Out.bolClamping.map;
END_IF
END_METHOD

METHOD Refill
VAR_INPUT
	intNbOfLDS: INT;
END_VAR
VAR
	/// Loop variable
	ii: INT;
END_VAR
// Simulation
fbSimulationTimer.PT := UDINT_TO_TIME(1000);
IF (CIf.SwCfg.bolSimulation) THEN
	// Cyclicle input into the top stopperbuffer
	fbSimulationTimer(); // set time/reset timer
	IF fbSimulationTimer.Q = TRUE THEN
		fbSimulationTimer.IN := FALSE;
	ELSE
		fbSimulationTimer.IN := TRUE;
	END_IF
			
END_IF

// Method refill 
CASE intSubState[intNbOfLDS] OF
	cSTA_SUB_WaitForJob: // LDS needs hanger
		IF (a_bolLDSNeedsHanger[intNbOfLDS]) THEN
			IF (p_fbSLB^.CtrlCIf^.Info.p_aCIf[intNbOfLDS]^.job.intState = 6)THEN //	Just open if PreStopper is closed
				a_pMultiChildCIF[intNbOfLDS]^.Job.intACmd:= Base_Elements.VLV_CmdState.cCMD_OPEN;
				udiTimeInStateRefill_ms[intNbOfLDS] := 0;
				intSubState[intNbOfLDS] := cSTA_SUB_WaitOpen;
			END_IF
		END_IF
	
	cSTA_SUB_WaitOpen:	// Waiting time between STB closing and junction opening
		udiTimeInStateRefill_ms[intNbOfLDS]:= udiTimeInStateRefill_ms[intNbOfLDS] + me.FUBInfo.udiSample_ms;
		IF (udiTimeInStateRefill_ms[intNbOfLDS] > SIf.Par.udiWaitingTime_ms) THEN
			intSubState[intNbOfLDS] := cSTA_SUB_Open;
		END_IF
		
	cSTA_SUB_Open:	
		IF (a_bolLDSNeedsHanger[intNbOfLDS] = 0) THEN
			intSubState[intNbOfLDS] := cSTA_SUB_WaitClose;
		END_IF
		
	cSTA_SUB_WaitClose:	// Waiting time between STB closing and junction closing
		IF (p_fbSLB^.CtrlCIf^.Info.p_aCIf[intNbOfLDS]^.job.intState = 6)THEN //	Just close if PreStopper is closed
			udiTimeInStateRefill_ms[intNbOfLDS] := 0;
			intSubState[intNbOfLDS] := cSTA_SUB_Close;
		END_IF
		
	cSTA_SUB_Close:
		udiTimeInStateRefill_ms[intNbOfLDS]:= udiTimeInStateRefill_ms[intNbOfLDS] + me.FUBInfo.udiSample_ms;
		IF (udiTimeInStateRefill_ms[intNbOfLDS] > SIf.Par.udiWaitingTime_ms) THEN
			a_pMultiChildCIF[intNbOfLDS]^.Job.intACmd:= Base_Elements.VLV_CmdState.cCMD_Close;
			intSubState[intNbOfLDS] := cSTA_SUB_WaitForJob;
		END_IF
END_CASE
END_METHOD

METHOD PROTECTED sta_OFF : BOOL
// state implemetation
//--------------------------------------------------------------------------------------
// Entry action
	IF (me.StateMachine.intState<>me.StateMachine.intStateLastCycle) THEN
		me.StateMachine.intStateLastCycle := me.StateMachine.intState;
		
	END_IF


//--------------------------------------------------------------------------------------
// Cyclic action
	IF (me.StateMachine.intState=me.StateMachine.intStateLastCycle) THEN
		
		;
		
		// State Change Condition
		IF me.intCmd=cCMD_RUN THEN
			me.StateMachine.intStateNext :=  cSTA_RUNBusy;
		END_IF
	END_IF




//--------------------------------------------------------------------------------------
// Exit action
	IF (me.StateMachine.intState<>me.StateMachine.intStateNext) THEN
		;
	END_IF
END_METHOD

METHOD PROTECTED sta_RUN : BOOL
VAR
	intNbOfLDS: INT;
END_VAR
// state implemetation
//--------------------------------------------------------------------------------------
// Entry action
	IF (me.StateMachine.intState<>me.StateMachine.intStateLastCycle) THEN
		me.StateMachine.intStateLastCycle := me.StateMachine.intState;
		
		//fbSimulationTimer.IN := FALSE;
		//fbSimulationTimer.PT := UDINT_TO_TIME(SIf.Par.udi_pulseTimeout_ms/10);
		//fbSimulationTimer(); // set time/reset timer
		//fbSimulationTimer.IN := TRUE; // start timer
		FOR intNbOfLDS := 0 TO cuintMaxStation DO
			intSubState[intNbOfLDS] := 500;	// Init Refill Substate
		END_FOR
	END_IF


//--------------------------------------------------------------------------------------
// Cyclic action
	IF (me.StateMachine.intState=me.StateMachine.intStateLastCycle) THEN
		
		// Simulation
		IF (CIf.SwCfg.bolSimulation) THEN
			//fbSimulationTimer(); // simulation time
			//IF (fbSimulationTimer.Q) THEN
			//	SIf.In.bolPulse.intern := NOT SIf.In.bolPulse.intern; // toggle pulse
			//	fbSimulationTimer.IN := FALSE;
			//ELSE
			//	fbSimulationTimer.IN := TRUE;
			//END_IF
		END_IF
		
		//IF NOT(pSLB_SIf^.Cur.bolBufferFull) THEN
		//	pStopperBuffer_CIf^.Job.intACmd := STB_CmdState.cCMD_RELEASE;
		//END_IF
		FOR intNbOfLDS := 0 TO cuintMaxStation DO
			IF (SIf.Par.a_bolEnableJunction[intNbOfLDS]) AND (a_pMultiChildCtrl[intNbOfLDS]<>0) THEN
				Refill(intNbOfLDS);
			END_IF
		END_FOR
		
		// State Change Condition
		IF me.intCmd=cCMD_OFF THEN
			me.StateMachine.intStateNext := cSTA_OFFBusy;
		END_IF
		
	END_IF



//--------------------------------------------------------------------------------------
// Exit action
	IF (me.StateMachine.intState<>me.StateMachine.intStateNext) THEN
		;
	END_IF
END_METHOD

METHOD PROTECTED sta_RUNBusy : BOOL
// state implemetation
//--------------------------------------------------------------------------------------
// Entry action
	IF (me.StateMachine.intState<>me.StateMachine.intStateLastCycle) THEN
		me.StateMachine.intStateLastCycle := me.StateMachine.intState;
		
		pTlpDrive_CIf^.Job.intACmd := cCMD_RUN;
		pSLB_CIf^.Job.intACmd := Base_PLC.cCMD_RUN;
		
	END_IF


//--------------------------------------------------------------------------------------
// Cyclic action
	IF (me.StateMachine.intState=me.StateMachine.intStateLastCycle) THEN
		
		// State Change Condition
		IF (pTlpDrive_CIf^.Job.intState = cSTA_RUN) THEN
			me.StateMachine.intStateNext := cSTA_RUN;
		END_IF
	END_IF



//--------------------------------------------------------------------------------------
// Exit action
	IF (me.StateMachine.intState<>me.StateMachine.intStateNext) THEN
		;
	END_IF
END_METHOD

METHOD PROTECTED StateMachine : BOOL
SUPER^.StateMachine();

// main statemachine of base controller
CASE me.StateMachine.intState OF
	 cSTA_RUN: 
        THIS^.sta_RUN();
	cSTA_RUNBusy:
        THIS^.sta_RUNBusy();
END_CASE;
END_METHOD

END_FUNCTION_BLOCK

// POUs/Controller/Lvl2/HPS (Heat Press Shirt Station)/FB_DtChnToLine_ChargeDone
FUNCTION_BLOCK FB_DtChnToLine_ChargeDone
VAR_INPUT
	bolResetError: BOOL;
	pSIf: POINTER TO T_Ctrl_SIf_HPS;
END_VAR
VAR_OUTPUT
	///Error value
	intError: INT;
END_VAR
VAR
	/// Internal Variable
	intStatemachine: INT;
	/// Data not correct
	bolDataBad: BOOL;
	/// Retry Counts for error message
	intCountRetry: INT;
	/// Buffer for Senddata
	aBuffer: ARRAY[0..cDtChnBuffer] OF T_ChargeDone_DtChn;
	/// Pointer for new Input
	intPBufferInput: INT;
	/// Pointer for readout
	intPBufferOutput: INT;
	/// Data Channel Specific Variable
	intIndexOldest: INT;
	/// Date and time of the oldes imput
	dtOldestTag: DT;
	fbGetSystemTime: GETSYSTEMTIME;
	stfileTime: T_FILETIME;
	dtActualTime: DT;
END_VAR
VAR CONSTANT
	cDtChnBuffer: INT := 20;
	cSTA_SUB_Data_Init: INT := 900;
	cSTA_SUB_Data_WaitForJob: INT := 902;
	cSTA_SUB_Data_SendData: INT := 904;
	cSTA_SUB_Data_Acknowledge: INT := 906;
	cSTA_SUB_Data_Retry: INT := 908;
	cSTA_SUB_Data_Error: INT := 910;
	cDataState_DONE: INT := -1;
	cDataState_Ready: INT := 1;
	cDataState_Retry: INT := -99;
	cDataState_Error: INT := -100;
	cMAX_RETRY: INT := 10;
	/// Error Codes
	cERR_BufferFull: INT := -99;
	cERR_NoSIF: INT := -100;
END_VAR

(*__________________________________________________________________________________________________
¦	
¦	Vistaprint Schweiz GmbH
¦	CH - 8401 Winterthur
¦
¦	www.vistaprint.ch - info@vistaprint.ch
¦___________________________________________________________________________________________________

Function desription:
Datachannel to send data to Lince Controller
Insert new Job with Method Creat in a Buffer
Send buffer elements if Linecontroller is ready


History:
Version		Date			Author		Comment
---------------------------------------------------------------------------------------------------
0.00.1		26.08.2013		AVM/PRE		Start history


___________________________________________________________________________________________________*)

// Data Channel to Receive Data from Line Controller
// Startup check States
IF (pSIf <> 0) THEN
	IF (intStatemachine < cSTA_SUB_Data_Init) THEN
		intStatemachine := cSTA_SUB_Data_Init;
	END_IF
ELSE
	intError := cERR_NoSIF;
END_IF

CASE intStatemachine OF
	cSTA_SUB_Data_Init:
		IF pSIf^.DtChnToLine.stChargeDone.intDataState = cDataState_DONE THEN
			intStatemachine := cSTA_SUB_Data_WaitForJob;
		END_IF
		
	cSTA_SUB_Data_WaitForJob:
		// New data arrived
		IF intPBufferInput <> intPBufferOutput THEN
			IF pSIf^.DtChnToLine.stChargeDone.intDataState = cDataState_DONE THEN
				intStatemachine := cSTA_SUB_Data_SendData;
			END_IF
		END_IF
	
	cSTA_SUB_Data_SendData:	
		pSIf^.DtChnToLine.stChargeDone.intLine := aBuffer[intPBufferOutput].intLine;
		pSIf^.DtChnToLine.stChargeDone.dtTimestamp := aBuffer[intPBufferOutput].dtTimestamp;
		pSIf^.DtChnToLine.stChargeDone.intDataState := cDataState_Ready;
		intStatemachine := cSTA_SUB_Data_Acknowledge;	
		
	cSTA_SUB_Data_Acknowledge:	
		IF pSIf^.DtChnToLine.stChargeDone.intDataState = cDataState_DONE THEN
			// Data read from Line Controller
			// Reset Buffer Element
			aBuffer[intPBufferOutput].dtTimestamp := DINT_TO_DT(0);
			aBuffer[intPBufferOutput].intDataState := 0;
			aBuffer[intPBufferOutput].intLine := 0;
			// Increase Read out pointer
			IF intPBufferOutput < cDtChnBuffer THEN
				intPBufferOutput := intPBufferOutput + 1;
			ELSE
				intPBufferOutput := 0;
			END_IF
			intStatemachine := cSTA_SUB_Data_WaitForJob;
			
		ELSIF pSIf^.DtChnToLine.stChargeDone.intDataState = cDataState_Retry THEN
			intStatemachine := cSTA_SUB_Data_Retry;
		ELSIF pSIf^.DtChnToLine.stChargeDone.intDataState = cDataState_Error THEN
			intStatemachine := cSTA_SUB_Data_Error;
		END_IF
		
	cSTA_SUB_Data_Retry:
			IF intCountRetry < cMAX_RETRY THEN
				intCountRetry := intCountRetry + 1;
				intStatemachine := cSTA_SUB_Data_SendData;
			ELSE
				intStatemachine := cSTA_SUB_Data_Error;
			END_IF

	cSTA_SUB_Data_Error:
		intError := intCountRetry;
		IF bolResetError = TRUE THEN
			intStatemachine := cSTA_SUB_Data_WaitForJob;
		END_IF
			
END_CASE

METHOD Creat : INT
VAR_INPUT
	In_intLine: INT;
END_VAR
// Insert a new Job to send at Line controller
// Only insert the job, if the buffer is not full, next input dosn't cross input and Outputpointer

// Get Systemtime
fbGetSystemTime(timeLoDW=>stfileTime.dwLowDateTime, timeHiDW=>stfileTime.dwHighDateTime);
dtActualTime := FILETIME_TO_DT( stfileTime );

IF ((intPBufferInput + 1) = intPBufferOutput) OR ((intPBufferInput = cDtChnBuffer) AND (intPBufferOutput = 0)) THEN
	Creat := cERR_BufferFull;
ELSE
	aBuffer[intPBufferInput].intLine := In_intLine;
	aBuffer[intPBufferInput].dtTimestamp := dtActualTime;
	IF intPBufferInput < cDtChnBuffer THEN
		intPBufferInput := intPBufferInput + 1;
	ELSE
		intPBufferInput := 0;
	END_IF
	Creat := intPBufferInput;
END_IF
END_METHOD

END_FUNCTION_BLOCK

